TYPE "LBP_typeAxisX"
TITLE = Axis interface / Interface d'axe
// User data type for blocks LBP_Axis1 [DB31] .. LBP_Axis31 [DB61] / Type de données utilisateur pour les blocs LBP_Axis1 [DB31] .. LBP_Axis31 [DB61]
   STRUCT
      A_FD_OR : Byte;   // Feedrate override / Correction d'avance
      A_DriveEnable : Bool;   // Drive test movement enable / Débloquer le déplacement pour test d'entraînement
      A_AckFixedStop : Bool;   // Acknowledge fixed stop reached / Acquittement accostage de butée
      A_SensorFixedStop : Bool;   // Sensor fixed stop / Détecteur butée
      A_ASpDisable : Bool;   // Axis/spindle disable / Désactiver axe/broche
      A_Follow_upMode : Bool;   // Follow-up mode / Mode poursuite
      A_PosMeas1 : Bool;   // Position measuring system 1 / Système de mesure de position 1
      A_PosMeas2 : Bool;   // Position measuring system 2 / Système de mesure de position 2
      A_ORactive : Bool;   // Override active / Correction active
      A_SWCam : Bool;   // SW cam activation / Activation came logicielle
      A_ContrEnable : Bool;   // Controller enable / Activer la commande
      A_DelDTGSpReset : Bool;   // Delete distance to go/Spindle-Reset / Effacer la distance restante à parcourir / Reset broche
      A_Clamp : Bool;   // Clamping in progress / Serrage en cours
      A_RefVal1 : Bool;   // Reference point value 1 / Valeur de point de référence 1
      A_RefVal2 : Bool;   // Reference point value 2 / Valeur de point de référence 2
      A_RefVal3 : Bool;   // Reference point value 3 / Valeur de point de référence 3
      A_RefVal4 : Bool;   // Reference point value 4 / Valeur de point de référence 4
      A_ExtZO : Bool;   // Import external ZO / Importer ZO externes
      A_EnabTravFixedStop : Bool;   // Enable travel to fixed stop / Activer déplacement pour accostage de butée
      A_FixedFD1 : Bool;   // Activate fixed feedrate 1 / Activer l'avance fixe 1
      A_FixedFD2 : Bool;   // Activate fixed feedrate 2 / Activer l'avance fixe 2
      A_FixedFD3 : Bool;   // Activate fixed feedrate 3 / Activer l'avance fixe 3
      A_FixedFD4 : Bool;   // Activate fixed feedrate 4 / Activer l'avance fixe 4
      A_VelocSpeedLimit : Bool;   // Velocity/spindle speed limitation / Limitation vitesse / vitesse de broche
      A_PrgtestAxRel : Bool;   // Program test axis/spindle release / Débloquer test de programme axe/broche
      A_HW1 : Bool;   // Activate handwheel 1 / Activer manivelle 1
      A_HW2 : Bool;   // Activate handwheel 2 / Activer manivelle 2
      A_HW3 : Bool;   // Activate handwheel 3 / Activer manivelle 3
      A_FDSpStop : Bool;   // Feed stop/spindle stop / Arrêt avance / arrêt broche
      A_Disable : Bool;   // Traversing key disable / Désactiver la touche de déplacement
      A_RapidTrOR : Bool;   // Rapid traverse override / Correction marche rapide
      A_Minus : Bool;   // Traversing key minus / Touche de déplacement moins
      A_Plus : Bool;   // Traversing key plus / Touche de déplacement plus
      A_INC1 : Bool;   // INC1
      A_INC10 : Bool;   // INC10
      A_INC100 : Bool;   // INC100
      A_INC1000 : Bool;   // INC1000
      A_INC10000 : Bool;   // INC10000
      A_INCVar : Bool;   // INC variable / Variable INC
      A_ContManTravel : Bool;   // Continuous manual travel / Mode manuel continu
      f5_7 : Bool;
      A_OEMAxis : Byte;   // OEM axis signals / Signaux des axes OEM
      A_InvHWDirOfRot : Bool;   // Inverting handwheel direction of rotation / Inverser sens de rotation manivelle
      f7_1 : Bool;
      f7_2 : Bool;
      f7_3 : Bool;
      f7_4 : Bool;
      f7_5 : Bool;
      f7_6 : Bool;
      f7_7 : Bool;
      A_NCASpChanA : Bool;   // Assign NC axis/spindle channel A / Affecter axe/broche CN au canal A
      A_NCASpChanB : Bool;   // Assign NC axis/spindle channel B / Affecter axe/broche CN au canal B
      A_NCASpChanC : Bool;   // Assign NC axis/spindle channel C / Affecter axe/broche CN au canal C
      A_NCASpChanD : Bool;   // Assign NC axis/spindle channel D / Affecter axe/broche CN au canal D
      A_NCASpStrobe : Bool;   // Activation of assignment with pos. edge / Activation de l'affection sur font montant
      f8_5 : Bool;
      f8_6 : Bool;
      A_PLCASp : Bool;   // Request PLC axis/spindle / Demander axe/broche AP
      A_Para_A : Bool;   // Parameter block servo A / Bloc de paramètres servo A
      A_Para_B : Bool;   // Parameter block servo B / Bloc de paramètres servo B
      A_Para_C : Bool;   // Parameter block servo C / Bloc de paramètres servo C
      A_LockParSetDef : Bool;   // Lock parameter set definition from NC / Bloquer la définition de jeu de paramètre depuis CN
      f9_4 : Bool;
      f9_5 : Bool;
      f9_6 : Bool;
      f9_7 : Bool;
      A_REPOSDelay : Bool;   // REPOS DELAY
      f10_1 : Bool;
      f10_2 : Bool;
      f10_3 : Bool;
      f10_4 : Bool;
      f10_5 : Bool;
      f10_6 : Bool;
      f10_7 : Bool;
      A_StartBrakeTest : Bool;   // Start brake test / Démarrer test de frein
      f11_1 : Bool;
      f11_2 : Bool;
      f11_3 : Bool;
      f11_4 : Bool;
      f11_5 : Bool;
      f11_6 : Bool;
      f11_7 : Bool;
      A_HWLimitMinus : Bool;   // Hardware limit switch minus / Fin de course matériel moins
      A_HWLimitPlus : Bool;   // Hardware limit switch plus / Fin de course matériel plus
      A_SWLimit2Minus : Bool;   // 2nd software limit switch minus / 2e fin de course logiciel moins
      A_SWLimit2Plus : Bool;   // 2nd software limit switch plus / 2e fin de course logiciel plus
      A_ModuloLimitEn : Bool;   // Modulo limit enabled / Limite modulo activée
      f12_5 : Bool;
      f12_6 : Bool;
      A_DelayRef : Bool;   // Delay reference point approach / Retarder l'accostage de point de référence
      A_JogFixPPos0 : Bool;   // JogFixPointPos 0
      A_JogFixPPos1 : Bool;   // JogFixPointPos 1
      A_JogFixPPos2 : Bool;   // JogFixPointPos 2
      A_JogToPos : Bool;   // Jog to position / Mode JOG vers position
      f13_4 : Bool;
      f13_5 : Bool;
      f13_6 : Bool;
      f13_7 : Bool;
      A_ProgtestSuppress : Bool;   // Program test to suppress / Inhiber test de programme
      A_ProgtestActivate : Bool;   // Activate program test / Activer test de programme
      f14_2 : Bool;
      f14_3 : Bool;
      f14_4 : Bool;
      f14_5 : Bool;
      f14_6 : Bool;
      f14_7 : Bool;
      f15 : Byte;
      A_ActGearA : Bool;   // Current gear stage A / Rapport de transmission actuel A
      A_ActGearB : Bool;   // Current gear stage B / Rapport de transmission actuel B
      A_ActGearC : Bool;   // Current gear stage C / Rapport de transmission actuel C
      A_GearChangeOv : Bool;   // Gear has changed over / Réducteur a changé de rapport
      A_Sp1Syn : Bool;   // Re-synchronize spindle 1 / Resynchroniser broche 1
      A_Sp2Syn : Bool;   // Re-synchronize spindle 2 / Resynchroniser broche 2
      A_NoMonitorGear : Bool;   // No monitoring when changing gear / Aucune surveillance pendant le changement de rapport de réducteur
      A_DeleteS : Bool;   // Delete S value / Supprimer la valeur S
      A_FD_ORSp : Bool;   // Feedrate override for spindle valid / Correction d'avance pour broche valide
      f17_1 : Bool;
      f17_2 : Bool;
      f17_3 : Bool;
      A_Sp1SynP : Bool;   // Re-synchronize spindle 1 for positioning / Resynchroniser broche 1 pour positionnement
      A_Sp2SynP : Bool;   // Re-synchronize spindle 2 for positioning / Resynchroniser broche 2 pour positionnement
      A_M3M4Inv : Bool;   // Invert M3/M4 / Inverser M3/M4
      f17_7 : Bool;
      f18_0 : Bool;
      f18_1 : Bool;
      f18_2 : Bool;
      f18_3 : Bool;
      A_OscilPLC : Bool;   // Oscillation via PLC / Oscillation via AP
      A_OscilSpeed : Bool;   // Enable Oscillation / Activer oscillation
      A_SetRotDirectRight : Bool;   // Setpoint osci. direct. right / Consigne sens d'oscillation à droite
      A_SetRotDirectLeft : Bool;   // Setpoint osci. direct. left / Consigne sens d'oscillation à gauche
      A_SpOR : Byte;   // Spindle override / Correction broche
      f20_0 : Bool;
      A_RUEncQuStop : Bool;   // Run-up encoder quick stop / Générateur de rampe Arrêt rapide
      f20_2 : Bool;
      A_SpeedSetpSmooth : Bool;   // Speed setpoint smoothing / Lissage consigne de vitesse
      f20_4 : Bool;
      A_HoldBrakeToOpen : Bool;   // Holding brake open / Frein à l'arrêt desserré
      f20_6 : Bool;
      f20_7 : Bool;
      A_ParA : Bool;   // Parameter set selection A / Jeux de paramètres sélection A
      A_ParB : Bool;   // Parameter set selection B / Jeux de paramètres sélection B
      A_ParC : Bool;   // Parameter set selection C / Jeux de paramètres sélection C
      A_MotA : Bool;   // Motor selection A / Sélection moteur A
      A_MotB : Bool;   // Motor selection B / Sélection moteur B
      A_MotOK : Bool;   // Motor selected / Moteur sélectionné
      A_IntegratDisable : Bool;   // N controller integrator disable / Commande N Désactiver intégrateur
      A_PulseEnable : Bool;   // Pulse enable / Activer impulsions
      f22_0 : Bool;
      f22_1 : Bool;
      f22_2 : Bool;
      f22_3 : Bool;
      f22_4 : Bool;
      f22_5 : Bool;
      f22_6 : Bool;
      f22_7 : Bool;
      f23_0 : Bool;
      f23_1 : Bool;
      f23_2 : Bool;
      f23_3 : Bool;
      f23_4 : Bool;
      f23_5 : Bool;
      f23_6 : Bool;
      f23_7 : Bool;
      f24_0 : Bool;
      A_ControlAx : Bool;   // Control Axis / Axe pilote
      f24_2 : Bool;
      f24_3 : Bool;
      A_TorqComp : Bool;   // Torque compensation / Compensation de couple
      A_ChangSetpOutAss0 : Bool;   // Bit value for CTRLOUT_changed - Change setpoint output assignment / Valeur de bit pour CTRLOUT_changed - Modifier l'affectation de la sortie de consigne
      A_ChangSetpOutAss1 : Bool;   // Bit value for CTRLOUT_changed - Change setpoint output assignment / Valeur de bit pour CTRLOUT_changed - Modifier l'affectation de la sortie de consigne
      A_MS : Bool;   // Main/Sub: activate coupling / Maître/esclave : activer le couplage
      A_DynBComp : Bool;   // Dynamic backlash compensation activated / Compensation dynamique de jeu activée
      f25_1 : Bool;
      f25_2 : Bool;
      f25_3 : Bool;
      f25_4 : Bool;
      f25_5 : Bool;
      f25_6 : Bool;
      f25_7 : Bool;
      f26_0 : Bool;
      f26_1 : Bool;
      f26_2 : Bool;
      A_CompContr : Bool;   // Compensation controller On / Contrôleur de compensation MARCHE
      A_FollowAxOv : Bool;   // Enable following axis override / Activer la correction de l'axe asservi
      f26_5 : Bool;
      f26_6 : Bool;
      f26_7 : Bool;
      A_DEPMCS : Bool;   // Resume: DEPMCS / Continuer : DEPMCS
      A_DEPBCS : Bool;   // Resume: DEPBCS / Continuer : DEPBCS
      A_Corr : Bool;   // Resume: Corr / Continuer : corr
      A_HIAxMove : Bool;   // Resume: HIAxMove / Continuer : HIAxMove
      A_StopDEPMCS : Bool;   // Stop: DEPMCS / Arrêt : DEPMCS
      A_StopDEPBCS : Bool;   // Stop: DEPBCS / Arrêt : DEPBCS
      A_StopCorr : Bool;   // Stop: Corr / Arrêt : corr
      A_StopHIAxMove : Bool;   // Stop: HIAxMove / Arrêt : HIAxMove
      A_OscillAxExtRev : Bool;   // OscillAxExtReversal
      A_AxReset : Bool;   // AXRESET
      A_AxResume : Bool;   // AXRESUME
      A_SetRP : Bool;   // Set reversal point / Définir point d'inversion
      A_ChangeRP : Bool;   // Change reversal point / Modifier le point d'inversion
      A_StopRP : Bool;   // Stop at next reversal point / Arrêt sur point d'inversion suivant
      A_Stop : Bool;   // Stop / Arrêt
      A_PLCAxis : Bool;   // PLC checks axis / AP vérifie axe
      f29_0 : Bool;
      f29_1 : Bool;
      f29_2 : Bool;
      f29_3 : Bool;
      A_StartGantSynRun : Bool;   // Start gantry synchronization run / Démarrer l'opération de synchronisation Gantry
      A_NoAutoSync : Bool;   // No auto sync / Aucune sync auto
      f29_6 : Bool;
      f29_7 : Bool;
      A_StopSpindle : Bool;   // Stop spindle / Arrêt broche
      A_StartCW : Bool;   // Start spindle clockwise / Démarrer broche avec rotation horaire
      A_StartCCW : Bool;   // Start spindle counterclockwise / Démarrer broche avec rotation antihoraire
      A_AutoGearStep : Bool;   // Autom. gear step change / Chmnt. auto rapport transmission
      A_PosSpindle : Bool;   // Position spindle / Position de broche
      f30_5 : Bool;
      f30_6 : Bool;
      f30_7 : Bool;
      f31_0 : Bool;
      f31_1 : Bool;
      f31_2 : Bool;
      f31_3 : Bool;
      A_Resynchronize : Bool;   // Resynchronize / Resynchroniser
      A_DisSync : Bool;   // Disable synchronization / Désactiver la synchronisation
      A_Tracksync : Bool;   // Track synchronism / Tracer synchronisme
      A_DelSyncRunCorr : Bool;   // Deleting synchronous run correction / Suppression de la correction marche synchrone
      f32_0 : Bool;
      f32_1 : Bool;
      f32_2 : Bool;
      f32_3 : Bool;
      f32_4 : Bool;
      f32_5 : Bool;
      f32_6 : Bool;
      f32_7 : Bool;
      f33_0 : Bool;
      f33_1 : Bool;
      f33_2 : Bool;
      f33_3 : Bool;
      f33_4 : Bool;
      f33_5 : Bool;
      f33_6 : Bool;
      f33_7 : Bool;
      A_SI_SetpLimBit0 : Bool;   // Set point limitation Bit0 / Limitation de consigne Bit 0
      A_SI_SetpLimBit1 : Bool;   // Set point limitation Bit1 / Limitation de consigne Bit 1
      f34_2 : Bool;
      A_ActivateBrakeRampForSs2e : Bool;   // Brakes with NCK ramp on selection of SS2E (MD36959 MA_SAFE_BRAKE_RAMP_TIME) / Freinage avec rampe du NCK lors de la sélection de SS2E (MD36959 MA_SAFE_BRAKE_RAMP_TIME)
      f34_4 : Bool;
      f34_5 : Bool;
      f34_6 : Bool;
      f34_7 : Bool;
      f35 : Byte;
      f36 : Array[36..55] of Byte;
      A_FeedDriveCAxEng : Bool;   // Separate feed drive as C axis engaged / Entraînement d'avance séparé activé en tant qu'axe C
      A_SpSpeedDisp : Bool;   // Spindle speed display / Affichage vitesse de broche
      A_SpInsideClamp : Bool;   // Spindle inside clamping / Serrage interne broche
      f56_3 : Bool;
      f56_4 : Bool;
      f56_5 : Bool;
      f56_6 : Bool;
      f56_7 : Bool;
      f57 : Byte;
      f58 : Word;
      E_SpNA : Bool;   // Spindle/no axis / Broche / aucun axe
      E_NCU_Link : Bool;   // NCU_link active axis / NCU_link axe actif
      E_EncodFreq1 : Bool;   // Encoder limit frequency 1 exceeded / Fréquence limite capteur 1 dépassée
      E_EncodFreq2 : Bool;   // Encoder limit frequency 2 exceeded / Fréquence limite capteur 2 dépassée
      E_RefSyn1 : Bool;   // Referenced/synchronized 1 / Référencé/synchronisé 1
      E_RefSyn2 : Bool;   // Referenced/synchronized 2 / Référencé/synchronisé 2
      E_ExactCoarse : Bool;   // Position reached with exact stop coarse / Position atteinte avec arrêt précis approx.
      E_ExactFine : Bool;   // Position reached with exact stop fine / Position atteinte avec arrêt précis fin
      E_TravRequ : Bool;   // Travel request / Demande de déplacement
      E_AxialAlarm : Bool;   // Axial alarm / Alarme d'axe
      E_AxisReady : Bool;   // Axis ready / Axe prêt
      E_Follow_upMode : Bool;   // Follow-up mode active / Mode poursuite actif
      E_Stat : Bool;   // Axis/spindle stationary (n<nmin) / Axe/broche à l'arrêt (n<nmin)
      E_PositContr : Bool;   // Position controller active / Commande de positionnement active
      E_SpeedContr : Bool;   // Speed controller active / Régulateur de vitesse actif
      E_CurrentContr : Bool;   // Current controller active / Commande actuelle active
      E_SWCam : Bool;   // Software cams active / Came logicielle active
      E_HWOverlay : Bool;   // Handwheel overlay active / Superposition manivelle actif
      E_RevFD : Bool;   // Revolutional feedrate active / Avance par tour active
      E_MeasAct : Bool;   // Measuring active / Mesurage actif
      E_ActTravFStop : Bool;   // Activate travel to fixed stop / Activer déplacement pour accostage de butée
      E_FixedStop : Bool;   // Fixed stop reached / Butée atteinte
      E_ForceFixedStop : Bool;   // Force fixed stop limited / Force butée limitée
      E_AxContainerRot : Bool;   // Axis container rotation active / Conteneur d'axe Rotation activée
      E_AxReset : Bool;   // Axis reset done / Reset axe effectué
      E_PLCCtrlAx : Bool;   // PLC controlled axis / Axe commandé par AP
      E_AxStop : Bool;   // Axis stop active / Arrêt d'axe actif
      E_AxSpDisable : Bool;   // Axis/spindle disable active / Désactivation axe/broche active
      E_StopDEPMCS : Bool;   // Stop DEPMCS active / Arrêt DEPMCS actif
      E_StopDEPBCS : Bool;   // Stop DEPBCS active / Arrêt DEPBCS actif
      E_StopCorr : Bool;   // Stop Corr active / Arrêt corr actif
      E_StopHIAxMove : Bool;   // Stop HIAxMove active / Arrêt HIAxMove actif
      E_HW1 : Bool;   // Handwheel 1 active / Manivelle 1 active
      E_HW2 : Bool;   // Handwheel 2 active / Manivelle 2 active
      E_HW3 : Bool;   // Handwheel 3 active / Manivelle 3 active
      f64_3 : Bool;
      E_TReqMinus : Bool;   // Travel request minus / Demande de déplacement moins
      E_TReqPlus : Bool;   // Travel request plus / Demande de déplacement plus
      E_TCMinus : Bool;   // Traverse command minus / Instruction de déplacement moins
      E_TCPlus : Bool;   // Traverse command plus / Instruction de déplacement plus
      E_INC1 : Bool;   // INC1
      E_INC10 : Bool;   // INC10
      E_INC100 : Bool;   // INC100
      E_INC1000 : Bool;   // INC1000
      E_INC10000 : Bool;   // INC10000
      E_INCVar : Bool;   // INC variable / Variable INC
      E_ContManTravelAct : Bool;   // Continuous manual travel active / Mode manuel continu actif
      f65_7 : Bool;
      E_OEMAxis : Byte;   // OEM axis signals / Signaux des axes OEM
      E_InvHWDirOfRot : Bool;   // Handwheel direction of rotation invert actively / Inverser activement sens manivelle
      f67_1 : Bool;
      f67_2 : Bool;
      f67_3 : Bool;
      f67_4 : Bool;
      f67_5 : Bool;
      f67_6 : Bool;
      f67_7 : Bool;
      E_NCASpChanA : Bool;   // NC axis/spindle in channel A / Axe/broche CN dans canal A
      E_NCASpChanB : Bool;   // NC axis/spindle in channel B / Axe/broche CN dans canal B
      E_NCASpChanC : Bool;   // NC axis/spindle in channel C / Axe/broche CN dans canal C
      E_NCASpChanD : Bool;   // NC axis/spindle in channel D / Axe/broche CN dans canal D
      E_PLCType : Bool;   // New type requested by PLC / Nouveau type demandé de l'AP
      E_ChPoss : Bool;   // Change axis possible / Modification d'axe possible
      E_NeutrASp : Bool;   // Neutral axis/spindle / Axe/broche neutre
      E_PLCASp : Bool;   // PLC axis/spindle / Axe/broche AP
      E_ParS_A : Bool;   // Parameter block servo A / Bloc de paramètres servo A
      E_ParS_B : Bool;   // Parameter block servo B / Bloc de paramètres servo B
      E_ParS_C : Bool;   // Parameter block servo C / Bloc de paramètres servo C
      E_NCUNumLink_3 : Bool;
      E_NCUNumLink_4 : Bool;
      E_NCUNumLink_5 : Bool;
      E_NCUNumLink_6 : Bool;
      E_NCUNumLink_7 : Bool;
      E_ReposSh : Bool;   // REPOS shift / REPOS Décalage
      E_ReposShValid : Bool;   // REPOS shift valid / REPOS Décalage valide
      E_ReposDelayQuit : Bool;   // REPOS delay quit / REPOS Terminer temporisation
      f70_3 : Bool;
      f70_4 : Bool;
      E_SI_Drv_SICSCC : Bool;   // DRV-Safety Integrated with SIC/SCC active / DRV Safety Integrated avec SIC/SCC actif
      E_SI_Drv_Parameterized : Bool;   // Drive based Safety Intergated (SI) function enabled (at least one function in parameter "p9501" or "p9601" is parameterized) / Fonction Drive based Safety Integrated (SI) débloquée (au moins une fonction est paramétrée dans le paramètre "p9501" ou "p9601")
      f70_7 : Bool;
      E_BrakeTest : Bool;   // Brake test active / Test de frein actif
      f71_1 : Bool;
      f71_2 : Bool;
      f71_3 : Bool;
      E_POS_RESTORED1 : Bool;   // POS_RESTORED 1
      E_POS_RESTORED2 : Bool;   // POS_RESTORED 2
      f71_6 : Bool;
      E_PLCAxDedic : Bool;   // PLC axis dedicated / Axe AP dédié
      E_MMC_REPOSDelay : Bool;   // HMI REPOS DELAY
      f72_1 : Bool;
      f72_2 : Bool;
      f72_3 : Bool;
      f72_4 : Bool;
      f72_5 : Bool;
      f72_6 : Bool;
      f72_7 : Bool;
      f73 : Byte;
      f74_0 : Bool;
      f74_1 : Bool;
      f74_2 : Bool;
      f74_3 : Bool;
      E_ModLimEnAct : Bool;   // Modulo limit enabled active / Limite modulo activée actif
      f74_5 : Bool;
      f74_6 : Bool;
      f74_7 : Bool;
      E_JogFixPPos0Act : Bool;   // JogFixPointPos 0 active / JogFixPointPos 0 activé
      E_JogFixPPos1Act : Bool;   // JogFixPointPos 1 active / JogFixPointPos 1 activé
      E_JogFixPPos2Act : Bool;   // JogFixPointPos 2 active / JogFixPointPos 2 activé
      E_JogFixPPos0 : Bool;   // JogFixPointPos 0 reached / JogFixPointPos 0 atteint
      E_JogFixPPos1 : Bool;   // JogFixPointPos 1 reached / JogFixPointPos 1 atteint
      E_JogFixPPos2 : Bool;   // JogFixPointPos 2 reached / JogFixPointPos 2 atteint
      E_JogToPos : Bool;   // Jog to position active / Mode JOG vers position actif
      E_JogPos : Bool;   // Jog position reached / Position JOG atteinte
      E_ScratchPulse : Bool;   // Scratch pulse
      f76_1 : Bool;
      f76_2 : Bool;
      f76_3 : Bool;
      E_PathAxis : Bool;   // Path axis / Axe d'interpolation
      E_PosAxis : Bool;   // Positioning axis / Axe de positionnement
      E_IndexAxisPos : Bool;   // Indexing axis in position / Axe indexé en position
      E_CurvePos : Bool;   // Curve axis in position / Axe de contournage en position
      E_CollCheckRedSpeed : Bool;   // Reduced speed of Collisions Check / Vitesse réduite du contrôle de collision
      f77_1 : Bool;
      f77_2 : Bool;
      f77_3 : Bool;
      f77_4 : Bool;
      f77_5 : Bool;
      f77_6 : Bool;
      f77_7 : Bool;
      E_FPosAxis : Real;   // F function (REAL format) for positioning axes / Fonction F (format REAL) pour axes de positionnement
      E_SetpGearA : Bool;   // Setpoint gear stage A / Consigne de rapport de transmission A
      E_SetpGearB : Bool;   // Setpoint gear stage B / Consigne de rapport de transmission B
      E_SetpGearC : Bool;   // Setpoint gear stage C / Consigne de rapport de transmission C
      E_GearChange : Bool;   // Gear changeover / Changement de rapport réducteur
      f82_4 : Bool;
      f82_5 : Bool;
      f82_6 : Bool;
      f82_7 : Bool;
      E_SpeedLimit : Bool;   // Speed limit exceeded / Limite de vitesse dépassée
      E_SetSpeedLimit : Bool;   // Setpoint speed limited / Consigne de vitesse limitée
      E_SetSpeedIncreased : Bool;   // Setpoint speed increased / Consigne de vitesse augmentée
      E_GeoMonit : Bool;   // Geometry monitoring / Surveillance de géométrie
      E_SupportAreaViol : Bool;   // Support area limits violated / Limites de la zone de support dépassées
      E_SetRange : Bool;   // Spindle in setpoint range / Broche dans la plage consigne
      E_SpeedMonit : Bool;   // Speed monitoring / Surveillance de vitesse
      E_ActRotRight : Bool;   // Actual rotation direction right / Sens de rotation actuel horaire
      E_ConstCuttSpeed : Bool;   // Const. cutting speed active / Vitesse de coupe constante active
      E_SUG : Bool;   // SUG active (grinding wheel surface speed) / VPM active (vitesse périphérique de meule)
      E_CLG : Bool;   // CLG active / CLG actif
      E_Tapping : Bool;   // Tapping without compensating chuck / Taraudage sans porte-taraud compensateur
      E_SyncMode : Bool;   // Synchronous mode spindle active / Mode broche synchrone actif
      E_PosMode : Bool;   // Positioning mode spindle active / Mode positionnement broche actif
      E_OscillMode : Bool;   // Oscillation mode spindle active / Mode oscillation broche actif
      E_ContrMode : Bool;   // Control mode spindle active / Mode de commande broche actif
      E_ToolDynLimit : Bool;   // Tool with dynamics limit / Outil avec limite dynamique
      f85_1 : Bool;
      f85_2 : Bool;
      f85_3 : Bool;
      f85_4 : Bool;
      E_SpInPosition : Bool;   // Spindle in position / Broche en position
      f85_6 : Bool;
      f85_7 : Bool;
      E_MFunct : Int;   // M function (INT) for spindle / Fonction M (INT) pour broche
      E_SFunct : Real;   // S function (REAL) for spindle / Fonction S (REAL) pour broche
      f92_0 : Bool;
      E_RUEncDisabl : Bool;   // Run-up encoder disable active / Blocage codeur de démarrage actif
      f92_2 : Bool;
      E_SpeedSetpSmooth : Bool;   // Speed setpoint smoothing active / Lissage consigne de vitesse actif
      E_RLIact : Bool;   // RLI active / RLI actif
      E_HoldBrakeOpened : Bool;   // Holding brake opened / Frein à l'arrêt desserré
      f92_6 : Bool;
      E_DriveRunEn : Bool;   // Drive run enabled / Déplacement entraînement activé
      E_ParA : Bool;   // Active parameter set A / Jeux de paramètres actif A
      E_ParB : Bool;   // Active parameter set B / Jeux de paramètres actif B
      E_ParC : Bool;   // Active parameter set C / Jeux de paramètres actif C
      E_MotA : Bool;   // Active motor A / Moteur actif A
      E_MotB : Bool;   // Active motor B / Moteur actif B
      E_MotOK : Bool;   // Drive ready / Entraînement prêt
      E_IntegratDisable : Bool;   // N controller integrator disabled / Commande N Intégrateur désactivé
      E_PulseEnable : Bool;   // Pulses enabled / Impulsions débloquées
      E_MTempWarn : Bool;   // Prewarning motor temperature / Avertissement température moteur
      E_HTempWarn : Bool;   // Prewarning heat sink temperature / Avertissement température radiateur
      E_RUComplete : Bool;   // Ramp-up complete / Démarrage terminé
      E_MdMdx : Bool;   // Md<Mdx
      E_NactNmin : Bool;   // nact<nmin
      E_NactNx : Bool;   // nact<nx
      E_NactNset : Bool;   // nact=nset
      E_Message : Bool;   // Variable message function 1 / Fonction de signalisation variable 1
      E_UDClessAlThreshold : Bool;   // UDC-link < alarm threshold / Lien UDC < seuil d'alarme
      E_DcVoltageAlarmAct : Bool;   // ESR: DC link voltage is below the specified minimum / AER : la tension du circuit intermédiaire est inférieure au minimum spécifié
      E_GeneratorOperationAct : Bool;   // ESR: generator operation is active / AER : le fonctionnement du générateur est actif
      E_SpeedBelowMin : Bool;   // ESR: actual speed is below specified minimum speed - axis is a generator axis / AER : la vitesse réelle est inférieure à la vitesse minimale spécifiée – l'axe est un axe de générateur
      E_Message2 : Bool;   // Variable message function 2 / Fonction de signalisation variable 2
      E_Message3 : Bool;   // Variable message function 3 / Fonction de signalisation variable 3
      f95_6 : Bool;
      E_I2TLimit : Bool;   // Power Section I2T limit / Partie puissance limite I2T
      f96_0 : Bool;
      E_AxisCtrl : Bool;   // Axis control active / Commande d'axe active
      E_MSFine : Bool;   // Main/Sub: speed difference is within the fine tolerance range / Maître/esclave : la différence de vitesse se situe dans la plage de tolérance fine
      E_MSCoarse : Bool;   // Main/Sub: speed difference is within the coarse tolerance range / Maître/esclave : la différence de vitesse se situe dans la plage de tolérance grossière
      E_MSCompContr : Bool;   // Main/Sub: torque compensatory controller is active / Maître/esclave : le régulateur de compensation de couple est actif
      E_BitValCtrlOutChang0 : Bool;   // Bit value for CTRLOUT_changed 0: Change setpoint output assignment / Valeur de CTRLOUT_changed 0 : modifier l'affectation de sortie de consigne
      E_BitValCtrlOutChang1 : Bool;   // Bit value for CTRLOUT_changed 1: Change setpoint output assignment / Valeur de CTRLOUT_changed 1 : modifier l'affectation de sortie de consigne
      E_MS : Bool;   // Main/Sub: coupling is active / Maître/esclave : le couplage est actif
      f97 : Byte;
      E_SyncronFine : Bool;   // Synchronism fine / Synchronisme fin
      E_SyncronCoarse : Bool;   // Synchronism coarse / Synchronisme approx
      E_ActValCoupling : Bool;   // Actual value coupling / Valeur réelle couplage
      f98_3 : Bool;
      E_OverlayMotion : Bool;   // Overlaid motion / Mouvement superposé
      E_SWL : Bool;   // Speed warning limit reached / Valeur limite d'alarme pour vitesse atteinte
      E_AWL : Bool;   // Acceleration warning limit reached / Valeur limite d'alarme pour accélération atteinte
      E_EmRetr : Bool;   // Emergency retraction active / Retrait d'urgence actif
      E_MasterSp : Bool;   // Generic coupling: spindle is leading spindle / Couplage générique : la broche est une broche pilote
      E_SlaveSp : Bool;   // Generic coupling: spindle is following spindle / Couplage générique : la broche est une broche asservie
      E_SyncRunCorrDOut : Bool;   // Synchronous run correction driven out / Correction synchronisme dépassée
      E_AxisAccel : Bool;   // Axis accelerated / Axe accéléré
      E_Sync : Bool;   // Synchronization active / Synchronisation active
      E_MSR : Bool;   // Max. speed reached / Vitesse max. atteinte
      E_MAR : Bool;   // Max. acceleration reached / Accélération max. atteinte
      f99_7 : Bool;
      f100_0 : Bool;
      f100_1 : Bool;
      E_OscillAxExtRev : Bool;   // OscillAxExt Reversal active / OscillAxExt Inversion active
      E_StopOscill : Bool;   // Oscillation cannot start / Impossible de démarrer oscillation
      E_ErrorOscill : Bool;   // Error during oscillation / Erreur lors de l'oscillation
      E_SparkOut : Bool;   // Spark-out active / Passes à lécher actives
      E_OscillMotion : Bool;   // Oscillation motion active / Mouvement d'oscillation actif
      E_Oscill : Bool;   // Oscillation active
      f101_0 : Bool;
      f101_1 : Bool;
      E_GantCOLimit : Bool;   // Gantry cut-off limit exceeded / Limite coupure axe Gantry atteinte
      E_GantWarn : Bool;   // Gantry warning limit exceeded / Gantry Limite d'alarme dépassée
      E_SynRunStart : Bool;   // Synchronization run ready to start / Synchronisme prêt à démarrer
      E_GantGroupSyn : Bool;   // Gantry grouping is synchronous / Groupage Gantry synchronisé
      E_GantLeadAxis : Bool;   // Gantry leading axis / Axe pilote Gantry
      E_GantAxis : Bool;   // Gantry axis / Axe Gantry
      E_DynBComp : Bool;   // Dynamic backlash compensation activated / Compensation dynamique de jeu activée
      f102_1 : Bool;
      f102_2 : Bool;
      E_ClampTolerance : Bool;   // Clamp tolerance exceeded / Tolérance de serrage d'axe dépassée
      f102_4 : Bool;
      E_PosMeas1 : Bool;   // Position measuring system 1 active / Système de mesure de position 1 actif
      E_PosMeas2 : Bool;   // Position measuring system 2 active / Système de mesure de position 2 actif
      f102_7 : Bool;
      E_SyncRunCorrIncl : Bool;   // Synchronous run correction is included / Correction synchronisme incluse
      f103_1 : Bool;
      f103_2 : Bool;
      f103_3 : Bool;
      E_Syncron2Fine : Bool;   // Synchronism fine / Synchronisme fin
      E_Syncron2Coarse : Bool;   // Synchronism coarse / Synchronisme approx
      f103_6 : Bool;
      f103_7 : Bool;
      E_AIAxis : Array[1..31] of Bool;   // Active infeed axis[1..31] / Axe de pénétration active [1..31]
      f108_0 : Bool;
      f108_1 : Bool;
      f108_2 : Bool;
      f108_3 : Bool;
      f108_4 : Bool;
      f108_5 : Bool;
      f108_6 : Bool;
      f108_7 : Bool;
      f109_0 : Bool;
      f109_1 : Bool;
      f109_2 : Bool;
      f109_3 : Bool;
      f109_4 : Bool;
      f109_5 : Bool;
      f109_6 : Bool;
      f109_7 : Bool;
      f110_0 : Bool;
      f110_1 : Bool;
      f110_2 : Bool;
      f110_3 : Bool;
      f110_4 : Bool;
      f110_5 : Bool;
      f110_6 : Bool;
      f110_7 : Bool;
      f111_0 : Bool;
      f111_1 : Bool;
      f111_2 : Bool;
      f111_3 : Bool;
      f111_4 : Bool;
      f111_5 : Bool;
      f111_6 : Bool;
      f111_7 : Bool;
      f112 : Byte;
      f113 : Byte;
      f114 : Byte;
      f115 : Byte;
      f116 : Byte;
      f117_0 : Bool;
      f117_1 : Bool;
      f117_2 : Bool;
      f117_3 : Bool;
      f117_4 : Bool;
      f117_5 : Bool;
      f117_6 : Bool;
      f117_7 : Bool;
      f118 : DWord;
      f122 : DWord;
      f126 : Word;   // Internal / Interne
      E_MMC_ProgtestSuppress : Bool;   // HMI->PLC: Suppress program test / HMI ->AP : inhiber test de programme
      E_MMC_ProgtestActivate : Bool;   // HMI->PLC: Activate program test / HMI ->AP : activer test de programme
      f128_2 : Bool;
      f128_3 : Bool;
      f128_4 : Bool;
      f128_5 : Bool;
      f128_6 : Bool;
      f128_7 : Bool;
      f129 : Byte;
      E_FormatBit0DDS : Bool;   // Bit 0 for drive data set switchover (DDS) / Bit 0 pour la commutation du jeu de paramètres d'entraînement (DDS)
      E_FormatBit1DDS : Bool;   // Bit 1 for drive data set switchover (DDS) / Bit 1 pour la commutation du jeu de paramètres d'entraînement (DDS)
      E_FormatBit2DDS : Bool;   // Bit 2 for drive data set switchover (DDS) / Bit 2 pour la commutation du jeu de paramètres d'entraînement (DDS)
      E_FormatBit3DDS : Bool;   // Bit 3 for drive data set switchover (DDS) / Bit 3 pour la commutation du jeu de paramètres d'entraînement (DDS)
      E_FormatBit4DDS : Bool;   // Bit 4 for drive data set switchover (DDS) / Bit 4 pour la commutation du jeu de paramètres d'entraînement (DDS)
      f130_5 : Bool;
      f130_6 : Bool;
      E_MDS_DDS_InterfacesValid : Bool;   // Motor and drive data set interfaces invalid / Jeux de paramètres moteur et d'entraînement Interfaces valides
      f131 : Byte;
      E_SensorAv : Bool;   // Sensors available / Capteurs disponibles
      E_S1aMeasARod : Bool;   // Sensor S1: analogous measurement position of actuating rod / Capteur S1 : position de mesure analogique de la tige d'actionnement
      f132_2 : Bool;
      f132_3 : Bool;
      E_S4dPistonStopP : Bool;   // Sensor S4: digital value piston stop position / Capteur S4 : valeur numérique position d'arrêt piston
      E_S5dAngleShaft : Bool;   // Sensor S5: digital value angle situation shaft / Capteur S5 : valeur numérique position angulaire arbre
      E_S6Temp : Bool;   // Sensor S6: temperature / Capteur S6 : température
      f132_7 : Bool;
      f133 : Byte;
      E_ClampingState : Int;   // State of the clamping system / État du système de serrage
      E_AnalogSensor : Int;   // Analog sensor on the motor / Capteur analogique sur moteur
      f138_0 : Bool;
      f138_1 : Bool;
      f138_2 : Bool;
      f138_3 : Bool;
      E_S4PistonStopP : Bool;   // Sensor S4: piston stop position / Capteur S4 : position d'arrêt piston
      E_S5AngleShaft : Bool;   // Sensor S5: angle situation shaft / Capteur S5 : position angulaire arbre
      f138_6 : Bool;
      f138_7 : Bool;
      f139 : Byte;
      SCC : Struct   // PLC to Drive (SCC) / AP vers entraînement (SCC)
         CW1 : Struct
            TeststopStart : Bool;   // Test stops for extended functions / Stops pour test pour fonctions étendues
            res140_1 : Bool;
            res140_2 : Bool;
            res140_3 : Bool;
            res140_4 : Bool;
            CloseBrake : Bool;   // Close internal Brake / Serrer le frein interne
            res140_6 : Bool;
            res140_7 : Bool;
            res141 : Byte;
         END_STRUCT;
         CW3 : Struct
            res142 : Byte;
            SelectionSBT : Bool;   // Selection: safe brake test / Sélection : test de frein sûr
            BT_Start : Bool;   // Start: brake test / Démarrage : test de frein
            Brake_1_2 : Bool;   // Brake test with brake 1 or 2 / Test de frein avec frein 1 ou 2
            DirOfROT : Bool;   // Direction of rotation / Sens de rotation
            Testseq_1_2 : Bool;   // Test sequence 1 or 2 / Séquence de test 1 ou 2
            BrakeClosed : Bool;   // Feedback external brake / Signalisation en retour frein externe
            res143_6 : Bool;
            res143_7 : Bool;
         END_STRUCT;
      END_STRUCT;
      res144_163 : Array[144..163] of Byte;
      SIC : Struct   // Drive to PLC (SIC) / Entraînement vers AP (SIC)
         SW1 : Struct
            SLA_Sel : Bool;   // Safely Limited Acceleration selected / Accélération limitée sûre sélectionnée
            SLS_LimBit0_Sel : Bool;   // Safely-Limited Speed: limit Bit0 selected / Vitesse limitée sûre : limite bit0 sélectionnée
            SLS_LimBit1_Sel : Bool;   // Safely-Limited Speed: limit Bit1 selected / Vitesse limitée sûre : limite bit1 sélectionnée
            res164_3 : Bool;
            res164_4 : Bool;
            res164_5 : Bool;
            ESR_Req : Bool;   // Extended Stop and Retract requested / Arrêt étendu et retrait demandé
            SF_Message_Act : Bool;   // Safety error active / Erreur de sécurité active
            STO_Act : Bool;   // Safe torque off: active / Suppression sûre du couple : active
            SS1_Act : Bool;   // Safe Stop1: active / Stop sûr 1 : actif
            SS2_Act : Bool;   // Safe Stop2: active / Stop sûr 2 : actif
            SOS_Act : Bool;   // Safe Operating Stop: active / Arrêt de fonctionnement sûr : actif
            SLS_Act : Bool;   // Safely-Limited Speed: active / Vitesse limitée sûre : active
            SOS_Sel : Bool;   // Safe Operating Stop: selected / Arrêt de fonctionnement sûr : sélectionné
            SLS_Sel : Bool;   // Safely-Limited Speed: selected / Vitesse limitée sûre : sélectionnée
            InternalEvent : Bool;   // Safety error with Stop A active / Erreur de sécurité avec butée A active
         END_STRUCT;
         SW2 : Struct
            SDI_P_Sel : Bool;   // Safe direction positive: selected / Direction sûre positive : sélectionnée
            SDI_N_Sel : Bool;   // Safe direction negative: selected / Direction sûre négative : sélectionnée
            res166_2 : Bool;
            res166_3 : Bool;
            TestStopAct : Bool;   // Test stop active / Stop pour test actif
            TestStopReq : Bool;   // Test stop requested / Stop pour test demandé
            res166_6 : Bool;
            res166_7 : Bool;
            res167_0 : Bool;
            res167_1 : Bool;
            res167_2 : Bool;
            res167_3 : Bool;
            SLP_LimBit0_Sel : Bool;   // Safely-Limited Position: limit Bit0 selected / Position limitée sûre : limite bit0 sélectionnée
            res167_5 : Bool;
            res167_6 : Bool;
            SLP_Sel : Bool;   // Safely-Limited Position: selected / Position limitée sûre : sélectionnée
         END_STRUCT;
         V_Limit_B : DInt;   // Setpoint speed limit effective / Limite de consigne de vitesse active
         SW3 : Struct
            res172_0 : Bool;
            res172_1 : Bool;
            res172_2 : Bool;
            SS2E_ACTIVE : Bool;   // SS2E active / SS2E actif
            SS2ESR : Bool;   // SS2ESR active / SS2ESR actif
            res172_5 : Bool;
            AcceptSLPAct : Bool;   // Acceptance test Safely-Limited Position active / Essai de réception position limitée sûre : actif
            AcceptTestSel : Bool;   // Acceptance test selected / Essai de réception sélectionné
            SBT_Sel : Bool;   // Safety break test: selected / Test de frein de sécurité : sélectionné
            SetpSettingDrive : Bool;   // Setpoint input is in the drive during the SBT / L'entrée de consigne est dans l'entraînement pendant le SBT
            Brake_1_2 : Bool;   // Test with brake 1 or 2 / Test avec frein 1 ou 2
            BT_Act : Bool;   // Brake test: active / Test de frein : actif
            BT_OK : Bool;   // Brake test: OK / Test de frein : OK
            BT_Finished : Bool;   // Brake test: finished / Test de frein : terminé
            BrakeReq : Bool;   // External brake close requested / Serrage de frein externe demandé
            SignLoadTorque : Bool;   // Sign of load torque is negative / Signe couple de charge négatif
         END_STRUCT;
      END_STRUCT;
      res174_187 : Array[174..187] of Byte;
      CW7 : Struct
         ReservedBit08 : Bool;
         ReservedBit09 : Bool;
         ReservedBit10 : Bool;
         ReservedBit11 : Bool;
         ReservedBit12 : Bool;
         ReservedBit13 : Bool;
         ReservedBit14 : Bool;
         ReservedBit15 : Bool;
         A_DisablePowerReduction : Bool;   // DYNEGMA: disable power reduction / DYNEGMA : désactiver la réduction de puissance
         A_DisableCurrReduction : Bool;   // Motor overtemperature: disable current reduction / Surchauffe du moteur : désactiver la réduction de puissance
         ReservedBit02 : Bool;
         ReservedBit03 : Bool;
         ReservedBit04 : Bool;
         ReservedBit05 : Bool;
         ReservedBit06 : Bool;
         ReservedBit07 : Bool;
      END_STRUCT;
      SW7 : Struct
         E_EncMaintenanceRequired : Bool;   // Encoder maintenance required / Maintenance du codeur requise
         ReservedBit09 : Bool;
         ReservedBit10 : Bool;
         ReservedBit11 : Bool;
         ReservedBit12 : Bool;
         ReservedBit13 : Bool;
         ReservedBit14 : Bool;
         ReservedBit15 : Bool;
         E_TorqueLimited : Bool;   // DYNEGMA: torque limited / DYNEGMA : couple limité
         E_CurrReductionActive : Bool;   // Motor overtemperature: current reduction active / Surchauffe du moteur : réduction de puissance active
         E_MotorTempModelAlarm : Bool;   // Motor overtemperature: motor temperature model alarm active / Surchauffe du moteur : alarme de modèle thermique du moteur active
         E_PolePosIdentPassed : Bool;   // Pole position identification with encoder successfully carried out / Identification de la position des pôles avec codeur effectuée avec succès
         ReservedBit04 : Bool;
         ReservedBit05 : Bool;
         E_AndConditionFulfilled : Bool;   // AND logic operation: condition fulfilled / Opération logique ET : condition remplie
         E_OrConditionFulfilled : Bool;   // OR logic operation: condition fulfilled / Opération logique OU : condition remplie
      END_STRUCT;
   END_STRUCT;
END_TYPE

TYPE "LBP_typeChanX"
TITLE = Channel interface / Interface de canal
// User data type for blocks LBP_Chan1 [DB21] .. LBP_Chan10 [DB30] / Type de données utilisateur pour les blocs LBP_Chan1 [DB21] .. LBP_Chan10 [DB30]
   STRUCT
      f0_0 : Bool;
      f0_1 : Bool;
      f0_2 : Bool;
      A_DRF : Bool;   // Activate DRF / Activer DRF
      A_SBL : Bool;   // Activate single block / Activer bloc par bloc
      A_M01 : Bool;   // Activate M01 / Activer M01
      A_DRY : Bool;   // Activate dry run feedrate / Activer avance marche d'essai
      f0_7 : Bool;
      A_Ref : Bool;   // Activate referencing / Activer référencement
      A_ProtZone : Bool;   // Enable protection zones / Activer zones de protection
      A_SynOff : Bool;   // Synchronous action off / Action synchrone désactivée
      A_TM_TimOut : Bool;   // Activate time-out (TM) / Activer timeout (TM)
      A_CLC_Stop : Bool;   // CLC stop / Stop CLC
      A_CLC_OR : Bool;   // CLC override / Correction CLC
      A_PLC_ActCompl : Bool;   // PLC action completed / Action AP terminée
      A_ProgTest : Bool;   // Activate program test / Activer test de programme
      A_SKP0 : Bool;   // Activate skip block \0 / Activer ignorer bloc \0
      A_SKP1 : Bool;   // Activate skip block \1 / Activer ignorer bloc \1
      A_SKP2 : Bool;   // Activate skip block \2 / Activer ignorer bloc \2
      A_SKP3 : Bool;   // Activate skip block \3 / Activer ignorer bloc \3
      A_SKP4 : Bool;   // Activate skip block \4 / Activer ignorer bloc \4
      A_SKP5 : Bool;   // Activate skip block \5 / Activer ignorer bloc \5
      A_SKP6 : Bool;   // Activate skip block \6 / Activer ignorer bloc \6
      A_SKP7 : Bool;   // Activate skip block \7 / Activer ignorer bloc \7
      A_StrokEnab : Bool;   // Stroke enable / Activer course
      A_ManStrokEnab : Bool;   // Manual stroke enable / Activation manuelle de la course
      A_StrokSup : Bool;   // Stroke suppression / Inhibition de course
      A_StrokDelayed : Bool;   // Stroke delayed / Course retardée
      A_StrokStop : Bool;   // Stroke not operating / Course inopérante
      A_ManRelStroke2 : Bool;   // Manual release of stroke 2 / Déblocage manuel de la course 2
      A3_6 : Bool;
      A3_7 : Bool;
      A_FD_OR : Byte;   // Feedrate override / Correction d'avance
      A_RT_OR : Byte;   // Rapid traverse override / Correction marche rapide
      A_FDdisable : Bool;   // Feed disable / Désactiver avance
      A_RIdisable : Bool;   // Read-in disable / Désactiver importation
      A_DeleteDTG : Bool;   // Delete distance to go / Effacer la distance restante à parcourir
      A_SP_Clear : Bool;   // Delete UP number of passes / Supprimer nombre UP de passes
      A_ProgAbort : Bool;   // Program level abort / Abandon niveau de programme
      A_F_Limit : Bool;   // Tool path feedrate limitation / Trajectoire d'outil limitation d'avance
      A_RT_ORA : Bool;   // Rapid traverse override active / Correction marche rapide active
      A_FD_ORA : Bool;   // Feedrate override active / Correction d'avance active
      A_NCStartDisabl : Bool;   // NC start disable / Désactiver Départ CN
      A_NCStart : Bool;   // NC start / Départ CN
      A_NCStopBlock : Bool;   // NC stop at block limit / Arrêt CN à la limite de bloc
      A_NCStop : Bool;   // NC stop / Arrêt CN
      A_NCStopASp : Bool;   // NC stop axes plus spindle / Arrêt CN axes et broche
      A_SuppStartLock : Bool;   // Suppress Start Lock / Inhiber blocage de démarrage
      A_CfgStopFunc : Bool;   // Activate configured stop function / Activer la fonction d'arrêt configuré
      A_Reset : Bool;   // Reset
      A_MRP : Array[1..10] of Bool;   // Activate machine-related protection zone [1..10] / Activer zone de protection référencée dans le SCM [1..10]
      A_CSP : Array[1..10] of Bool;   // Activate channel-specific protection zone [1..10] / Activer zone de protection spécifique au canal [1..10]
      A_Geo : Array[1..3] of Struct   // Control signals for geometry axis [1..3] / Signaux de commande pour axe géométrique [1..3]
         HW1 : Bool;   // Activate handwheel 1 / Activer manivelle 1
         HW2 : Bool;   // Activate handwheel 2 / Activer manivelle 2
         HW3 : Bool;   // Activate handwheel 3 / Activer manivelle 3
         FDStop : Bool;   // Feedrate stop / Arrêt avance
         Disabl : Bool;   // Traversing key disable / Désactiver la touche de déplacement
         RapidTrOR : Bool;   // Rapid traverse override / Correction marche rapide
         Minus : Bool;   // Traversing key minus / Touche de déplacement moins
         Plus : Bool;   // Traversing key plus / Touche de déplacement plus
         INC1 : Bool;   // INC 1
         INC10 : Bool;   // INC 10
         INC100 : Bool;   // INC 100
         INC1000 : Bool;   // INC 1000
         INC10000 : Bool;   // INC 10000
         INCVar : Bool;   // INC variable / Variable INC
         ContManTravel : Bool;   // Continuous manual travel / Mode manuel continu
         f1_7 : Bool;
         OEM : Byte;   // OEM signals / Signaux OEM
         InvHWDirOfRot : Bool;   // Invert handwheel direction of rotation / Inverser sens de rotation manivelle
         f3_1 : Bool;
         f3_2 : Bool;
         f3_3 : Bool;
         f3_4 : Bool;
         f3_5 : Bool;
         f3_6 : Bool;
         f3_7 : Bool;
      END_STRUCT;
      f24_0 : Bool;
      E_MMC_CfgStopFunc : Bool;   // HMI: configured stop function (CST) is selected / IHM : La fonction d'arrêt configuré (CST) est sélectionnée
      E_MMC_AtStopSetOvrZero : Bool;   // HMI: Set to 0% for stop override / IHM : à l'arrêt, régler la correction sur 0 %
      E_MMC_DRF : Bool;   // HMI DRF selected / HMI DRF sélectionné
      E_MMC_M01AssocNC : Bool;   // Select M01 associated with NC / Sélectionner M01 associé à CN
      E_MMC_M01 : Bool;   // HMI M01 selected / HMI M01 sélectionné
      E_MMC_DRY : Bool;   // HMI Dry-run feedrate selected / HMI Marche d'essai avance sélectionnée
      f24_7 : Bool;
      E_MMC_REPOSPM_0 : Bool;   // HMI REPOSPATHMODE 0
      E_MMC_REPOSPM_1 : Bool;   // HMI REPOSPATHMODE 1
      E_MMC_REPOSPM_2 : Bool;   // HMI REPOSPATHMODE 2
      E_MMC_FD_OR4RT_OR : Bool;   // HMI Feedrate override for rapid traverse selected / HMI Correction d'avance marche rapide sélectionnée
      E_MMC_REPOSMode : Bool;   // HMI REPOS MODE EDGE
      f25_5 : Bool;
      f25_6 : Bool;
      E_MMC_ProgTest : Bool;   // Program test selected / Test de programme sélectionné
      E_MMC_SKP0 : Bool;   // HMI skip block selected \0 / HMI Ignorer bloc sélectionné \0
      E_MMC_SKP1 : Bool;   // HMI skip block selected \1 / HMI Ignorer bloc sélectionné \1
      E_MMC_SKP2 : Bool;   // HMI skip block selected \2 / HMI Ignorer bloc sélectionné \2
      E_MMC_SKP3 : Bool;   // HMI skip block selected \3 / HMI Ignorer bloc sélectionné \3
      E_MMC_SKP4 : Bool;   // HMI skip block selected \4 / HMI Ignorer bloc sélectionné \4
      E_MMC_SKP5 : Bool;   // HMI skip block selected \5 / HMI Ignorer bloc sélectionné \5
      E_MMC_SKP6 : Bool;   // HMI skip block selected \6 / HMI Ignorer bloc sélectionné \6
      E_MMC_SKP7 : Bool;   // HMI skip block selected \7 / HMI Ignorer bloc sélectionné \7
      E_MMC_SKP8 : Bool;   // HMI skip block selected \8 / HMI Ignorer bloc sélectionné \8
      E_MMC_SKP9 : Bool;   // HMI skip block selected \9 / HMI Ignorer bloc sélectionné \9
      f27_2 : Bool;
      f27_3 : Bool;
      f27_4 : Bool;
      f27_5 : Bool;
      f27_6 : Bool;
      f27_7 : Bool;
      A_OEM : Byte;
      A_FixedFD1 : Bool;   // Activate fixed feedrate 1 / Activer l'avance fixe 1
      A_FixedFD2 : Bool;   // Activate fixed feedrate 2 / Activer l'avance fixe 2
      A_FixedFD3 : Bool;   // Activate fixed feedrate 3 / Activer l'avance fixe 3
      A_FixedFD4 : Bool;   // Activate fixed feedrate 4 / Activer l'avance fixe 4
      A_PTP_Travel : Bool;   // Activate PTP traversal / Activer déplacement PTP
      A_DisablWP_Counter : Bool;   // Deactivate workpiece counter / Désactiver compteur de pièces
      A_DisablWearMon : Bool;   // Deactivate wear monitoring / Désactiver surveillance d'usure
      A_DontDisablTool : Bool;   // Do not disable tool / Ne pas désactiver outil
      A_ContHW1 : Bool;   // Activate contour handwheel 1 / Activer manivelle de contour 1
      A_ContHW2 : Bool;   // Activate contour handwheel 2 / Activer manivelle de contour 2
      A_ContHW3 : Bool;   // Activate contour handwheel 3 / Activer manivelle de contour 3
      A_ContHWsim : Bool;   // Simulated contour handwheel on / Manivelle de contour simulée Marche
      A_ContHWneg : Bool;   // Contour handwheel neg. route / Manivelle de contour dépl. nég.
      A_NCKrelatedM01 : Bool;   // Activate NCK-related M01 / Activer M01 relatif à la NCK
      A_JOG_Circles : Bool;   // JOG in circles / JOG en cercles
      A_NoToolChangeCmd : Bool;   // No tool change commands / Aucun ordre de changement d'outil
      A_REPOSPM_0 : Bool;   // REPOSPATHMODE 0
      A_REPOSPM_1 : Bool;   // REPOSPATHMODE 1
      A_REPOSPM_2 : Bool;   // REPOSPATHMODE 2
      f31_3 : Bool;
      A_REPOSMode : Bool;   // REPOS MODE EDGE
      A_InvCHWDirOfRot : Bool;   // Inverting contour handwheel direction of rotation / Inversion du sens de rotation de la manivelle
      A_SKP8 : Bool;   // Activate skip block \8 / Activer ignorer bloc \8
      A_SKP9 : Bool;   // Activate skip block \9 / Activer ignorer bloc \9
      E_ExecExtern : Bool;   // Execution from external source active / Exécution à partir de source externe active
      f32_1 : Bool;
      f32_2 : Bool;
      E_ActBlock : Bool;   // Action block active / Bloc d'action actif
      E_BegBlock : Bool;   // Approach block active / Bloc d'accostage actif
      E_M01 : Bool;   // M0/M1 active / M0/M1 actif
      E_LastActBlock : Bool;   // Last action block active / Dernier bloc d'action actif
      f32_7 : Bool;
      E_Ref : Bool;   // Referencing active / Référencement actif
      E_OrieToolholder : Bool;   // Orientable toolholder active / Porte-outil orientable actif
      E_RevFD : Bool;   // Revolutional feedrate active / Avance par tour active
      E_HWOverlay : Bool;   // Handwheel override active / Correction manivelle active
      E_BlockSearch : Bool;   // Block search active / Recherche de blocs active
      E_M30 : Bool;   // M2/M30 active / M2/M30 actif
      E_Transform : Bool;   // Transformation active
      E_ProgTest : Bool;   // Program test active / Test de programme actif
      E_OEMChan : Byte;   // OEM channel signals feedback / Signalisation en retour signaux de canal OEM
      E_ProgRunning : Bool;   // Program running / Programme en cours d'exécution
      E_ProgWait : Bool;   // Program waiting / Programme en attente
      E_ProgStop : Bool;   // Program stopped / Programme arrêté
      E_ProgInterrupt : Bool;   // Program interrupted / Programme interrompu
      E_ProgAborted : Bool;   // Program aborted / Programme abandonné
      E_ChanActive : Bool;   // Channel active / Canal actif
      E_ChanInterrupt : Bool;   // Channel interrupted / Canal interrompu
      E_ChanReset : Bool;   // Channel reset / Reset canal
      E_StartReq : Bool;   // Start request / Demande de démarrage
      E_StopReq : Bool;   // Stop request / Demande d'arrêt
      E_AxesRef : Bool;   // All axes referenced / Référencer tous les axes
      E_AxesStop : Bool;   // All axes stationary / Tous les axes à l'arrêt
      E_IR_Activ : Bool;   // Interrupt processing active / Traitement d'interruption actif
      E_ChanRO : Bool;   // Channel ready for operation / Canal prêt à fonctionner
      E_NCKalarmChan : Bool;   // Channel-specific NCK alarm present / Alarme NCK spécifique à un canal présente
      E_NCKalarmStop : Bool;   // NCK alarm with processing stop present / Alarme NCK avec d'arrêt d'usinage présente
      E_CHW1 : Bool;   // Contour handwheel 1 on / Manivelle de contour 1
      E_CHW2 : Bool;   // Contour handwheel 2 on / Manivelle de contour 2
      E_CHW3 : Bool;   // Contour handwheel 3 on / Manivelle de contour 3
      E_CLC : Bool;   // CLC active / CLC actif
      E_CLCStopLL : Bool;   // CLC stopped lower limit / CLC arrêté limite inférieure
      E_CLCStopUL : Bool;   // CLC stopped upper limit / CLC arrêté limite supérieure
      E_RIEnabIgnored : Bool;   // Read-in enable is ignored / Activation Charger ignorée
      E_StopBlkEndSBLsuppr : Bool;   // Stop at block end with SBL is suppressed / Inhiber arrêt sur fin de bloc avec SBL
      E_StrokeEA : Bool;   // Stroke release active / Déblocage course actif
      E_AcknManStrokEnab : Bool;   // Acknowledgment of manual stroke release / Acquittement déblocage manuel de course
      f38_2 : Bool;
      f38_3 : Bool;
      f38_4 : Bool;
      f38_5 : Bool;
      f38_6 : Bool;
      f38_7 : Bool;
      E_ProtZoneNOK : Bool;   // Protection zones not guaranteed / Zones de protection non garanties
      E_NCalarmWithProgStop : Bool;   // NC alarm with program stop / Alarme CN avec arrêt du programme
      f39_2 : Bool;
      E_ReducedDynamicsActive : Bool;   // Reduced dynamics mode is active / Le mode de dynamique réduite est actif
      E_SblStopAtBlockEnd : Bool;   // Stop at block end due to single block / Arrêt en fin de bloc en raison du mode bloc par bloc
      E_InvCHWDirOfRot : Bool;   // Contour handwheel direction of rotation invert actively / Inversion active du sens de rotation manivelle de contour
      E_CfgStopFuncActive : Bool;   // Configured stop function is activated / La fonction d'arrêt configuré est activée
      E_CfgStopAtBlockEnd : Bool;   // Stop at block end due to configured stop / Arrêt en fin de bloc en raison de l'arrêt configuré
      E_Geo : Array[1..3] of Struct   // Status signals of geometry axis [1..3] / Signaux d'état de l'axe géométrique [1..3]
         HW1 : Bool;   // Handwheel 1 active / Manivelle 1 active
         HW2 : Bool;   // Handwheel 2 active / Manivelle 2 active
         HW3 : Bool;   // Handwheel 3 active / Manivelle 3 active
         f0_3 : Bool;
         TReqMinus : Bool;   // Travel requests minus / Demandes de déplacement moins
         TReqPlus : Bool;   // Travel requests plus / Demandes de déplacement plus
         TCMinus : Bool;   // Traverse command minus / Instruction de déplacement moins
         TCPlus : Bool;   // Traverse command plus / Instruction de déplacement plus
         INC1 : Bool;   // INC 1 active
         INC10 : Bool;   // INC 10 active
         INC100 : Bool;   // INC 100 active
         INC1000 : Bool;   // INC 1000 active
         INC10000 : Bool;   // INC 10000 active
         INCVar : Bool;   // INC variable active / Variable INC active
         ContManTravelAct : Bool;   // Continuous manual travel active / Mode manuel continu actif
         f1_7 : Bool;
         OEM : Byte;   // OEM signals / Signaux OEM
         InvHWDirOfRot : Bool;   // Handwheel direction of rotation invert actively / Inverser activement sens manivelle
         f3_1 : Bool;
         f3_2 : Bool;
         f3_3 : Bool;
         f3_4 : Bool;
         f3_5 : Bool;
         f3_6 : Bool;
         f3_7 : Bool;
         f4 : Byte;
      END_STRUCT;
      M1Change : Bool;   // M function 1 change / Fonction M 1 modification
      M2Change : Bool;   // M function 2 change / Fonction M 2 modification
      M3Change : Bool;   // M function 3 change / Fonction M 3 modification
      M4Change : Bool;   // M function 4 change / Fonction M 4 modification
      M5Change : Bool;   // M function 5 change / Fonction M 5 modification
      f58_5 : Bool;
      f58_6 : Bool;
      f58_7 : Bool;
      M1NDec : Bool;   // M function 1 not decoded / Fonction M 1 non décodée
      M2NDec : Bool;   // M function 2 not decoded / Fonction M 2 non décodée
      M3NDec : Bool;   // M function 3 not decoded / Fonction M 3 non décodée
      M4NDec : Bool;   // M function 4 not decoded / Fonction M 4 non décodée
      M5NDec : Bool;   // M function 5 not decoded / Fonction M 5 non décodée
      f59_5 : Bool;
      f59_6 : Bool;
      f59_7 : Bool;
      S1Change : Bool;   // S function 1 change / Fonction S 1 modification
      S2Change : Bool;   // S function 2 change / Fonction S 2 modification
      S3Change : Bool;   // S function 3 change / Fonction S 3 modification
      f60_3 : Bool;
      S1Quick : Bool;   // S function 1 quick / Fonction S 1 rapide
      S2Quick : Bool;   // S function 2 quick / Fonction S 2 rapide
      S3Quick : Bool;   // S function 3 quick / Fonction S 3 rapide
      f60_7 : Bool;
      T1Change : Bool;   // T function 1 change / Fonction T 1 modification
      T2Change : Bool;   // T function 2 change / Fonction T 2 modification
      T3Change : Bool;   // T function 3 change / Fonction T 3 modification
      f61_3 : Bool;
      T1Quick : Bool;   // T function 1 quick / Fonction T 1 rapide
      T2Quick : Bool;   // T function 2 quick / Fonction T 2 rapide
      T3Quick : Bool;   // T function 3 quick / Fonction T 3 rapide
      f61_7 : Bool;
      D1Change : Bool;   // D function 1 change / Fonction D 1 modification
      D2Change : Bool;   // D function 2 change / Fonction D 2 modification
      D3Change : Bool;   // D function 3 change / Fonction D 3 modification
      f62_3 : Bool;
      D1Quick : Bool;   // D function 1 quick / Fonction D 1 rapide
      D2Quick : Bool;   // D function 2 quick / Fonction D 2 rapide
      D3Quick : Bool;   // D function 3 quick / Fonction D 3 rapide
      f62_7 : Bool;
      EChange : Bool;   // E function change / Fonction E modification
      f63_1 : Bool;
      f63_2 : Bool;
      f63_3 : Bool;
      EQuick : Bool;   // E function quick / Fonction E rapide
      f63_5 : Bool;
      f63_6 : Bool;
      f63_7 : Bool;
      H1Change : Bool;   // H function 1 change / Fonction H 1 modification
      H2Change : Bool;   // H function 2 change / Fonction H 2 modification
      H3Change : Bool;   // H function 3 change / Fonction H 3 modification
      f64_3 : Bool;
      H1Quick : Bool;   // H function 1 quick / Fonction H 1 rapide
      H2Quick : Bool;   // H function 2 quick / Fonction H 2 rapide
      H3Quick : Bool;   // H function 3 quick / Fonction H 3 rapide
      f64_7 : Bool;
      F1Change : Bool;   // F function 1 change / Fonction F 1 modification
      F2Change : Bool;   // F function 2 change / Fonction F 2 modification
      F3Change : Bool;   // F function 3 change / Fonction F 3 modification
      F4Change : Bool;   // F function 4 change / Fonction F 4 modification
      F5Change : Bool;   // F function 5 change / Fonction F 5 modification
      F6Change : Bool;   // F function 6 change / Fonction F 6 modification
      f65_6 : Bool;
      f65_7 : Bool;
      M1Quick : Bool;   // M function 1 quick / Fonction M 1 rapide
      M2Quick : Bool;   // M function 2 quick / Fonction M 2 rapide
      M3Quick : Bool;   // M function 3 quick / Fonction M 3 rapide
      M4Quick : Bool;   // M function 4 quick / Fonction M 4 rapide
      M5Quick : Bool;   // M function 5 quick / Fonction M 5 rapide
      f66_5 : Bool;
      f66_6 : Bool;
      f66_7 : Bool;
      F1Quick : Bool;   // F function 1 quick / Fonction F 1 rapide
      F2Quick : Bool;   // F function 2 quick / Fonction F 2 rapide
      F3Quick : Bool;   // F function 3 quick / Fonction F 3 rapide
      F4Quick : Bool;   // F function 4 quick / Fonction F 4 rapide
      F5Quick : Bool;   // F function 5 quick / Fonction F 5 rapide
      F6Quick : Bool;   // F function 6 quick / Fonction F 6 rapide
      f67_6 : Bool;
      f67_7 : Bool;
      ExtM1 : Int;   // Extended address M function 1 (16 bit INT) / Fonction M à adresse étendue 1 (16 bits INT)
      M1 : DInt;   // M function 1 (DInt) / Fonction M 1 (DInt)
      ExtM2 : Int;   // Extended address M function 1 (16 bit INT) / Fonction M à adresse étendue 1 (16 bits INT)
      M2 : DInt;   // M function 2 (DInt) / Fonction M 2 (DInt)
      ExtM3 : Int;   // Extended address M function 1 (16 bit INT) / Fonction M à adresse étendue 1 (16 bits INT)
      M3 : DInt;   // M function 3 (DInt) / Fonction M 3 (DInt)
      ExtM4 : Int;   // Extended address M function 1 (16 bit INT) / Fonction M à adresse étendue 1 (16 bits INT)
      M4 : DInt;   // M function 4 (DInt) / Fonction M 4 (DInt)
      ExtM5 : Int;   // Extended address M function 1 (16 bit INT) / Fonction M à adresse étendue 1 (16 bits INT)
      M5 : DInt;   // M function 5 (DInt) / Fonction M 5 (DInt)
      ExtS1 : Int;   // Extended address S function 1 (16 bit INT) / Fonction S à adresse étendue 1 (16 bits INT)
      S1 : Real;   // S function 1 (REAL) / Fonction S 1 (REAL)
      ExtS2 : Int;   // Extended address S function 2 (16 bit INT) / Fonction S à adresse étendue 2 (16 bits INT)
      S2 : Real;   // S function 2 (REAL) / Fonction S 2 (REAL)
      ExtS3 : Int;   // Extended address S function 3 (16 bit INT) / Fonction S à adresse étendue 3 (16 bits INT)
      S3 : Real;   // S function 3 (REAL) / Fonction S 3 (REAL)
      ExtT1 : Int;   // Extended address T function 1 (16 bit INT)T : DINT; //T function (DInt)f122 : INT;f124 : INT;f126 : INT; //Change in case of 8-digit T function / Fonction T à adresse étendue 1 (16 Bit INT)T : DINT; //fonction T (DInt)f122 : INT;f124 : INT;f126 : INT; //Modifier pour une fonction T à 8 chiffres
      T1 : Int;   // T function 1 (INT) / Fonction T 1 (INT)
      ExtT2 : Int;   // Extended address T function 2 (16 bit INT) / Fonction T à adresse étendue 2 (16 bits INT)
      T2 : Int;   // T function 2 (INT) / Fonction T 2 (INT)
      ExtT3 : Int;   // Extended address T function 3 (16 bit INT) / Fonction T à adresse étendue 3 (16 bits INT)
      T3 : Int;   // T function 3 (INT) / Fonction T 3 (INT)
      ExtD1 : Byte;   // Extended address D function 1 (8 bit INT)D : INT;f132 : INT; //Change in case of 5-digit D function / Fonction D à adresse étendue 1 (8 bits INT)D : INT;f132 : INT; //Modifier pour une fonction D à 5 chiffres
      D1 : Byte;   // D function 1 (8 bit INT) / Fonction D 1 (8 bits INT)
      ExtD2 : Byte;   // Extended address D function 2 (8 bit INT) / Fonction D à adresse étendue 2 (8 bits INT)
      D2 : Byte;   // D function 2 (8 bit INT) / Fonction D 2 (8 bits INT)
      ExtD3 : Byte;   // Extended address D function 3 (8 bit INT) / Fonction D à adresse étendue 3 (8 bits INT)
      D3 : Byte;   // D function 3 (8 bit INT) / Fonction D 3 (8 bits INT)
      ExtE : Int;   // Extended address D function 3 (16 bit INT) / Fonction D à adresse étendue 3 (16 bits INT)
      "E" : Real;   // E function (REAL) / Fonction E (REAL)
      ExtH1 : Int;   // Extended address H function 1 (16 bit INT) / Fonction H à adresse étendue 1 (16 bits INT)
      H1 : Real;   // H function 1 (REAL), DInt also in DBD396 / Fonction H 1 (REAL), DInt également dans DBD396
      ExtH2 : Int;   // Extended address H function 2 (16 bit INT) / Fonction H à adresse étendue 2 (16 bits INT)
      H2 : Real;   // H function 2 (REAL), DInt also in DBD400 / Fonction H 2 (REAL), DInt également dans DBD400
      ExtH3 : Int;   // Extended address H function 3 (16 bit INT) / Fonction H à adresse étendue 3 (16 bits INT)
      H3 : Real;   // H function 3 (REAL), DInt also in DBD404 / Fonction H 3 (REAL), DInt également dans DBD404
      ExtF1 : Int;   // Extended address F function 1 (16 bit INT) / Fonction F à adresse étendue 1 (16 bits INT)
      F1 : Real;   // F function 1 (REAL) / Fonction F 1 (REAL)
      ExtF2 : Int;   // Extended address F function 2 (16 bit INT) / Fonction F à adresse étendue 2 (16 bits INT)
      F2 : Real;   // F function 2 (REAL) / Fonction F 2 (REAL)
      ExtF3 : Int;   // Extended address F function 3 (16 bit INT) / Fonction F à adresse étendue 3 (16 bits INT)
      F3 : Real;   // F function 3 (REAL) / Fonction F 3 (REAL)
      ExtF4 : Int;   // Extended address F function 4 (16 bit INT) / Fonction F à adresse étendue 4 (16 bits INT)
      F4 : Real;   // F function 4 (REAL) / Fonction F 4 (REAL)
      ExtF5 : Int;   // Extended address F function 5 (16 bit INT) / Fonction F à adresse étendue 5 (16 bits INT)
      F5 : Real;   // F function 5 (REAL) / Fonction F 5 (REAL)
      ExtF6 : Int;   // Extended address F function 6 (16 bit INT) / Fonction F à adresse étendue 6 (16 bits INT)
      F6 : Real;   // F function 6 (REAL) / Fonction F 6 (REAL)
      MDyn : Array[0..99] of Bool;   // Dynamic M functions [0..99] / Fonctions M dynamiques [0..99]
      GAct : Array[1..64] of Byte;   // Active G function of group [1..64] / Fonction G active du groupe [1..64]
      E_MRPactivated : Array[1..10] of Bool;   // Machine-related protection zone [1..10] preactivated / Zone de protection référencée dans le SCM [1..10] préactivé
      E_CSPactivated : Array[1..10] of Bool;   // Channel-specific protection zone [1..10] preactivated / Zone de protection spécifique au canal [1..10] préactivée
      E_MRPViolated : Array[1..10] of Bool;   // Machine-related protection zone [1..10] violated / Zone de protection référencée dans le SCM [1..10] dépassée
      E_CSPViolated : Array[1..10] of Bool;   // Channel-specific protection zone [1..10] violated from P4 on / Zone de protection spécifique au canal [1..10] dépassée à partir de P4
      f_280_0 : Bool;
      A_Str_Synon : Bool;   // Request of syn.action to NCK / Demande d'action synchrone vers NCK
      f_280_2 : Bool;
      f_280_3 : Bool;
      f_280_4 : Bool;
      f_280_5 : Bool;
      f_280_6 : Bool;
      f_280_7 : Bool;
      f_281_0 : Bool;
      A_Str_Synfrom : Bool;   // Request syn.action from NCK / Demande d'action synchrone depuis NCK
      f_281_2 : Bool;
      f_281_3 : Bool;
      f_281_4 : Bool;
      f_281_5 : Bool;
      f_281_6 : Bool;
      f_281_7 : Bool;
      f_282 : Int;
      f_284 : Int;
      f_286 : Int;
      f_288 : Int;
      f_290 : Int;
      f_292 : Int;
      f_294 : Int;
      f_296 : Int;
      f_298 : Int;
      A_SynDisabl : Array[1..64] of Bool;   // Disable synchronous actions / Désactiver actions synchrones
      E_SynDisabled : Array[1..64] of Bool;   // Synchronous actions disabled / Actions synchrones désactivées
      E_G00 : Bool;   // Active G functions / Fonctions G actives
      f316_1 : Bool;
      f316_2 : Bool;
      f316_3 : Bool;
      f316_4 : Bool;
      f316_5 : Bool;
      f316_6 : Bool;
      f316_7 : Bool;
      E_ExtLang : Bool;   // External language mode active / Mode de langage externe actif
      E_WS_Setp : Bool;   // Workpiece setpoint reached / Consigne pièce atteinte
      f317_2 : Bool;
      f317_3 : Bool;
      f317_4 : Bool;
      E_DriveTest : Bool;   // Travel request drive test / Demande de déplacement test d'entraînement
      E_PTP_Travel : Bool;   // PTP travel active / Déplacement PTP actif
      E_ToolMissing : Bool;   // Tool missing / Outil manquant
      E_ASUP_Stop : Bool;   // ASUP stopped / ASUP arrêté
      E_SearchAct : Bool;   // Search active / Recherche active
      E_TOFF : Bool;   // TOFF active / TOFF actif
      E_TOFFmovem : Bool;   // TOFF motion active / Déplacement TOFF actif
      E_StopDelayed : Bool;   // Stop delayed / Arrêt temporisé
      E_AssM01 : Bool;   // Associated M01 active / M01 associé actif
      E_DRY : Bool;   // Dry-run feedrate active / Marche d'essai avance active
      E_Overstore : Bool;   // Overstore active / Overstore actif
      E_REPOS_EdgeAckn : Bool;   // REPOS MODE EDGE ACKN
      E_REPOS_PMode0 : Bool;   // REPOS Path Mode Ackn 0
      E_REPOS_PMode1 : Bool;   // REPOS Path Mode Ackn 1
      E_REPOS_PMode2 : Bool;   // REPOS Path Mode Ackn 2
      E_DelayFTS : Bool;   // Delay FTS / Temporisation FTS
      E_REPOS_DEFERRA : Bool;   // REPOS DEFERRA L Chan
      E_Stop_NoDelayR : Bool;   // Stop-delay area not accepted / Plage de temporisation d'arrêt non acceptée
      E_NoToolChangeCmd : Bool;   // No tool change command active / Aucun ordre de changement d'outil actif
      A_Ori : Array[1..3] of Struct   // Control signals for orientation axes [1..3] / Signaux de commande pour axes d'orientation [1..3]
         HW1 : Bool;   // Activate handwheel 1 / Activer manivelle 1
         HW2 : Bool;   // Activate handwheel 2 / Activer manivelle 2
         HW3 : Bool;   // Activate handwheel 3 / Activer manivelle 3
         FDStop : Bool;   // Feedrate stop / Arrêt avance
         Disabl : Bool;   // Traversing key lock / Verrouiller touche de déplacement
         RapidTrOR : Bool;   // Rapid traverse override / Correction marche rapide
         Minus : Bool;   // Traversing key minus / Touche de déplacement moins
         Plus : Bool;   // Traversing key plus / Touche de déplacement plus
         INC1 : Bool;   // INC 1 active
         INC10 : Bool;   // INC 10 active
         INC100 : Bool;   // INC 100 active
         INC1000 : Bool;   // INC 1000 active
         INC10000 : Bool;   // INC 10000 active
         INCVar : Bool;   // INC variable active / Variable INC active
         OEM : Byte;   // OEM signals / Signaux OEM
         InvHWDirOfRot : Bool;   // Inverting handwheel direction of rotation / Inverser sens de rotation manivelle
         f3_1 : Bool;
         f3_2 : Bool;
         f3_3 : Bool;
         f3_4 : Bool;
         f3_5 : Bool;
         f3_6 : Bool;
         f3_7 : Bool;
      END_STRUCT;
      E_Ori : Array[1..3] of Struct   // Control signals for orientation axes [1..3] / Signaux de commande pour axes d'orientation [1..3]
         HW1 : Bool;   // Handwheel 1 active / Manivelle 1 active
         HW2 : Bool;   // Handwheel 2 active / Manivelle 2 active
         HW3 : Bool;   // Handwheel 3 active / Manivelle 3 active
         f0_3 : Bool;
         TReqMinus : Bool;   // Travel requests minus / Demandes de déplacement moins
         TReqPlus : Bool;   // Travel requests plus / Demandes de déplacement plus
         TCMinus : Bool;   // Traverse command minus / Instruction de déplacement moins
         TCPlus : Bool;   // Traverse command plus / Instruction de déplacement plus
         INC1 : Bool;   // INC 1 active
         INC10 : Bool;   // INC 10 active
         INC100 : Bool;   // INC 100 active
         INC1000 : Bool;   // INC 1000 active
         INC10000 : Bool;   // INC 10000 active
         INCVar : Bool;   // INC variable active / Variable INC active
         OEM : Byte;   // OEM signals / Signaux OEM
         InvHWDirOfRot : Bool;   // Handwheel direction of rotation invert actively / Inverser activement sens manivelle
         f3_1 : Bool;
         f3_2 : Bool;
         f3_3 : Bool;
         f3_4 : Bool;
         f3_5 : Bool;
         f3_6 : Bool;
         f3_7 : Bool;
      END_STRUCT;
      E_TPrewarnLimit : Bool;   // Tool prewarn limit reached / Seuil de préavis outil atteint
      E_TLimit : Bool;   // Tool limit reached / Limite d'outil atteinte
      E_TNewRepl : Bool;   // Transition to new replacement tool / Transition vers nouvel outil de remplacement
      E_TLastRepl : Bool;   // Last replacement tool of the tool group / Dernier outil de remplacement du groupe d'outils
      f344_4 : Bool;
      f344_5 : Bool;
      f344_6 : Bool;
      f344_7 : Bool;
      f345 : Byte;
      f346 : Byte;
      f347 : Byte;
      E_TNoPrewarnLimit : DInt;   // T number for tool prewarn limit / Numéro d'outil pour seuil de préavis outil
      E_TNoLimit : DInt;   // T number for tool limit / Numéro d'outil pour limite d'outil
      E_TNoNewRepl : DInt;   // T number of the new replacement tool / Numéro d'outil du nouvel outil de remplacement
      E_TNoLastRepl : DInt;   // T number of the last replacement tool / Numéro d'outil du dernier outil de remplacement
      E_Cycle_Sig : Array[0..15] of Bool;   // Cycles input signals / Signaux d'entrée des cycles
      A_Cycle_Sig : Array[0..15] of Bool;   // Cycles output signals / Signaux de sortie des cycles
      E_OEM_TechnoSig : Array[0..31] of Bool;   // OEM Techno input signals / Signaux d'entrée techno OEM
      A_OEM_TechnoSig : Array[0..31] of Bool;   // OEM Techno output signals / Signaux de sortie techno OEM
      E_ProgEvent_Start : Bool;   // Active Prog-Event: Start / Prog-Event actif : Démarrage
      E_ProgEvent_M30 : Bool;   // Active Prog-Event: M30 / Prog-Event actif : M30
      E_ProgEvent_Reset : Bool;   // Active Prog-Event: Start / Prog-Event actif : Démarrage
      E_ProgEvent_PowerOn : Bool;   // Active Prog-Event: Power on / Prog-Event actif : Mise sous tension
      E_ProgEvent_SearchRun : Bool;   // Active Prog-Event: Search / Prog-Event actif : Recherche
      f376_5 : Bool;
      f376_6 : Bool;
      f376_7 : Bool;
      E_CollCheckStop : Bool;   // Stop of Collision Check / Arrêt du contrôle de collision
      E_StopCondition : Bool;   // Stop Condition / Condition d'arrêt
      f377_2 : Bool;
      f377_3 : Bool;
      E_JogRetract : Bool;   // JOG Retract active / Retrait JOG actif
      E_RetractData : Bool;   // Retract data available / Données de retrait disponibles
      E_JOG_Circles : Bool;   // JOG in circles / JOG en cercles
      f377_7 : Bool;
      E_AnyAsup : Bool;   // AnyASUP activ / AnyASUP actif
      E_SilentAsup : Bool;   // Silent ASUP active / ASUP silencieux actif
      f378_2 : Bool;
      f378_3 : Bool;
      f378_4 : Bool;
      f378_5 : Bool;
      f378_6 : Bool;
      f378_7 : Bool;
      f379 : Byte;
      f380 : Array[0..31] of Bool;   // Reserved / Réservé
      A_ProgJump : Bool;   // Control program jump / Saut programme de commande
      f384_1 : Bool;
      f384_2 : Bool;
      f384_3 : Bool;
      f384_4 : Bool;
      f384_5 : Bool;
      f384_6 : Bool;
      f384_7 : Bool;
      A_InKeyG1 : Bool;   // Grinding signal 1 / Signal rectification 1
      A_InKeyG2 : Bool;   // Grinding signal 2 / Signal rectification 2
      A_InKeyG3 : Bool;   // Grinding signal 3 / Signal rectification 3
      A_InKeyG4 : Bool;   // Grinding signal 4 / Signal rectification 4
      A_InKeyG5 : Bool;   // Grinding signal 5 / Signal rectification 5
      A_InKeyG6 : Bool;   // Grinding signal 6 / Signal rectification 6
      A_InKeyG7 : Bool;   // Grinding signal 7 / Signal rectification 7
      A_InKeyG8 : Bool;   // Grinding signal 8 / Signal rectification 8
      A_InKeyGEn1 : Bool;   // Enable grinding signal 1 / Activer signal rectification 1
      A_InKeyGEn2 : Bool;   // Enable grinding signal 2 / Activer signal rectification 2
      A_InKeyGEn3 : Bool;   // Enable grinding signal 3 / Activer signal rectification 3
      A_InKeyGEn4 : Bool;   // Enable grinding signal 4 / Activer signal rectification 4
      A_InKeyGEn5 : Bool;   // Enable grinding signal 5 / Activer signal rectification 5
      A_InKeyGEn6 : Bool;   // Enable grinding signal 6 / Activer signal rectification 6
      A_InKeyGEn7 : Bool;   // Enable grinding signal 7 / Activer signal rectification 7
      A_InKeyGEn8 : Bool;   // Enable grinding signal 8 / Activer signal rectification 8
      A_InKeyGRunIn1 : Bool;   // Run grinding function 1 / Exécuter fonction de rectification 1
      A_InKeyGRunIn2 : Bool;   // Run grinding function 2 / Exécuter fonction de rectification 2
      A_InKeyGRunIn3 : Bool;   // Run grinding function 3 / Exécuter fonction de rectification 3
      A_InKeyGRunIn4 : Bool;   // Run grinding function 4 / Exécuter fonction de rectification 4
      A_InKeyGRunIn5 : Bool;   // Run grinding function 5 / Exécuter fonction de rectification 5
      A_InKeyGRunIn6 : Bool;   // Run grinding function 6 / Exécuter fonction de rectification 6
      A_InKeyGRunIn7 : Bool;   // Run grinding function 7 / Exécuter fonction de rectification 7
      A_InKeyGRunIn8 : Bool;   // Run grinding function 8 / Exécuter fonction de rectification 8
      E_TransformNo : Byte;   // Active transformation number / Numéro de la transformation active
      f389 : Byte;
      E_InKeyGIsEn1 : Bool;   // Grinding signal 1 enabled / Signal rectification 1 activé
      E_InKeyGIsEn2 : Bool;   // Grinding signal 2 enabled / Signal rectification 2 activé
      E_InKeyGIsEn3 : Bool;   // Grinding signal 3 enabled / Signal rectification 3 activé
      E_InKeyGIsEn4 : Bool;   // Grinding signal 4 enabled / Signal rectification 4 activé
      E_InKeyGIsEn5 : Bool;   // Grinding signal 5 enabled / Signal rectification 5 activé
      E_InKeyGIsEn6 : Bool;   // Grinding signal 6 enabled / Signal rectification 6 activé
      E_InKeyGIsEn7 : Bool;   // Grinding signal 7 enabled / Signal rectification 7 activé
      E_InKeyGIsEn8 : Bool;   // Grinding signal 8 enabled / Signal rectification 8 activé
      E_InKeyGRunOut1 : Bool;   // NCK status of grinding function 1 / État NCK fonction de rectification 1
      E_InKeyGRunOut2 : Bool;   // NCK status of grinding function 3 / État NCK fonction de rectification 3
      E_InKeyGRunOut3 : Bool;   // NCK status of grinding function 3 / État NCK fonction de rectification 3
      E_InKeyGRunOut4 : Bool;   // NCK status of grinding function 4 / État NCK fonction de rectification 4
      E_InKeyGRunOut5 : Bool;   // NCK status of grinding function 5 / État NCK fonction de rectification 5
      E_InKeyGRunOut6 : Bool;   // NCK status of grinding function 6 / État NCK fonction de rectification 6
      E_InKeyGRunOut7 : Bool;   // NCK status of grinding function 7 / État NCK fonction de rectification 7
      E_InKeyGRunOut8 : Bool;   // NCK status of grinding function 8 / État NCK fonction de rectification 8
      E_CART_JOG_MODE : Byte;   // Coordinate system for Cartesian jog traverse / Système de coordonnées pour déplacement cartésien en mode JOG
      f393 : Byte;
      f394 : Byte;
      f395 : Byte;
      H1_DInt : DInt;   // H Function 1 (DInt) / Fonction H 1 (DInt)
      H2_DInt : DInt;   // H Function 2 (DInt) / Fonction H 2 (DInt)
      H3_DInt : DInt;   // H Function 3 (DInt) / Fonction H 3 (DInt)
      E_AxisSelType : Byte;   // 0: MachAxis, 1: GeoAxis
      E_AxisSelAxis : Byte;   // Axis number / Numéro d'axe
      E_AxisSelRequest : Bool;   // Axis selection (touch) / Sélection d'axe (touche)
      f410_1 : Bool;
      f410_2 : Bool;
      f410_3 : Bool;
      f410_4 : Bool;
      f410_5 : Bool;
      f410_6 : Bool;
      f410_7 : Bool;
      f411 : Byte;
      A_AxisSelTypeActive : Byte;   // 0: MachAxis, 1: GeoAxis (return) / 0: MachAxis, 1: GeoAxis (retour)
      A_AxisSelAxisActive : Byte;   // Axis number (return) / Numéro d'axe (retour)
   END_STRUCT;
   // // A_Geo[2].HW1 : Activate handwheel 1 / Activer manivelle 1
   // // A_Geo[3].HW1 : Activate handwheel 1 / Activer manivelle 1
   // // A_Geo[2].HW2 : Activate handwheel 2 / Activer manivelle 2
   // // A_Geo[3].HW2 : Activate handwheel 2 / Activer manivelle 2
   // // A_Geo[2].HW3 : Activate handwheel 3 / Activer manivelle 3
   // // A_Geo[3].HW3 : Activate handwheel 3 / Activer manivelle 3
   // // A_Geo[2].FDStop : Feedrate stop / Arrêt avance
   // // A_Geo[3].FDStop : Feedrate stop / Arrêt avance
   // // A_Geo[2].Disabl : Traversing key disable / Désactiver la touche de déplacement
   // // A_Geo[3].Disabl : Traversing key disable / Désactiver la touche de déplacement
   // // A_Geo[2].RapidTrOR : Rapid traverse override / Correction marche rapide
   // // A_Geo[3].RapidTrOR : Rapid traverse override / Correction marche rapide
   // // A_Geo[2].Minus : Traversing key minus / Touche de déplacement moins
   // // A_Geo[3].Minus : Traversing key minus / Touche de déplacement moins
   // // A_Geo[2].Plus : Traversing key plus / Touche de déplacement plus
   // // A_Geo[3].Plus : Traversing key plus / Touche de déplacement plus
   // // A_Geo[2].INC1 : INC 1
   // // A_Geo[3].INC1 : INC 1
   // // A_Geo[2].INC10 : INC 10
   // // A_Geo[3].INC10 : INC 10
   // // A_Geo[2].INC100 : INC 100
   // // A_Geo[3].INC100 : INC 100
   // // A_Geo[2].INC1000 : INC 1000
   // // A_Geo[3].INC1000 : INC 1000
   // // A_Geo[2].INC10000 : INC 10000
   // // A_Geo[3].INC10000 : INC 10000
   // // A_Geo[2].INCVar : INC variable / Variable INC
   // // A_Geo[3].INCVar : INC variable / Variable INC
   // // A_Geo[2].ContManTravel : Continuous manual travel / Mode manuel continu
   // // A_Geo[3].ContManTravel : Continuous manual travel / Mode manuel continu
   // // A_Geo[2].OEM : OEM signals / Signaux OEM
   // // A_Geo[3].OEM : OEM signals / Signaux OEM
   // // A_Geo[2].InvHWDirOfRot : Invert handwheel direction of rotation / Inverser sens de rotation manivelle
   // // A_Geo[3].InvHWDirOfRot : Invert handwheel direction of rotation / Inverser sens de rotation manivelle
   // // A_Geo[1] : Control signals for geometry axis [1..3] / Signaux de commande pour axe géométrique [1..3]
   // // A_Geo[2] : Control signals for geometry axis [1..3] / Signaux de commande pour axe géométrique [1..3]
   // // A_Geo[3] : Control signals for geometry axis [1..3] / Signaux de commande pour axe géométrique [1..3]
   // // E_Geo[2].HW1 : Handwheel 1 active / Manivelle 1 active
   // // E_Geo[3].HW1 : Handwheel 1 active / Manivelle 1 active
   // // E_Geo[2].HW2 : Handwheel 2 active / Manivelle 2 active
   // // E_Geo[3].HW2 : Handwheel 2 active / Manivelle 2 active
   // // E_Geo[2].HW3 : Handwheel 3 active / Manivelle 3 active
   // // E_Geo[3].HW3 : Handwheel 3 active / Manivelle 3 active
   // // E_Geo[2].TReqMinus : Travel requests minus / Demandes de déplacement moins
   // // E_Geo[3].TReqMinus : Travel requests minus / Demandes de déplacement moins
   // // E_Geo[2].TReqPlus : Travel requests plus / Demandes de déplacement plus
   // // E_Geo[3].TReqPlus : Travel requests plus / Demandes de déplacement plus
   // // E_Geo[2].TCMinus : Traverse command minus / Instruction de déplacement moins
   // // E_Geo[3].TCMinus : Traverse command minus / Instruction de déplacement moins
   // // E_Geo[2].TCPlus : Traverse command plus / Instruction de déplacement plus
   // // E_Geo[3].TCPlus : Traverse command plus / Instruction de déplacement plus
   // // E_Geo[2].INC1 : INC 1 active
   // // E_Geo[3].INC1 : INC 1 active
   // // E_Geo[2].INC10 : INC 10 active
   // // E_Geo[3].INC10 : INC 10 active
   // // E_Geo[2].INC100 : INC 100 active
   // // E_Geo[3].INC100 : INC 100 active
   // // E_Geo[2].INC1000 : INC 1000 active
   // // E_Geo[3].INC1000 : INC 1000 active
   // // E_Geo[2].INC10000 : INC 10000 active
   // // E_Geo[3].INC10000 : INC 10000 active
   // // E_Geo[2].INCVar : INC variable active / Variable INC active
   // // E_Geo[3].INCVar : INC variable active / Variable INC active
   // E_Geo[1].ContManTravelAct := false;
   // // E_Geo[2].ContManTravelAct : Continuous manual travel active / Mode manuel continu actif
   // // E_Geo[3].ContManTravelAct : Continuous manual travel active / Mode manuel continu actif
   // E_Geo[1].f1_7 := false;
   // // E_Geo[2].OEM : OEM signals / Signaux OEM
   // // E_Geo[3].OEM : OEM signals / Signaux OEM
   // // E_Geo[2].InvHWDirOfRot : Handwheel direction of rotation invert actively / Inverser activement sens manivelle
   // // E_Geo[3].InvHWDirOfRot : Handwheel direction of rotation invert actively / Inverser activement sens manivelle
   // // E_Geo[1] : Status signals of geometry axis [1..3] / Signaux d'état de l'axe géométrique [1..3]
   // // E_Geo[2] : Status signals of geometry axis [1..3] / Signaux d'état de l'axe géométrique [1..3]
   // // E_Geo[3] : Status signals of geometry axis [1..3] / Signaux d'état de l'axe géométrique [1..3]
   // // A_Ori[2].HW1 : Activate handwheel 1 / Activer manivelle 1
   // // A_Ori[3].HW1 : Activate handwheel 1 / Activer manivelle 1
   // // A_Ori[2].HW2 : Activate handwheel 2 / Activer manivelle 2
   // // A_Ori[3].HW2 : Activate handwheel 2 / Activer manivelle 2
   // // A_Ori[2].HW3 : Activate handwheel 3 / Activer manivelle 3
   // // A_Ori[3].HW3 : Activate handwheel 3 / Activer manivelle 3
   // // A_Ori[2].FDStop : Feedrate stop / Arrêt avance
   // // A_Ori[3].FDStop : Feedrate stop / Arrêt avance
   // // A_Ori[2].Disabl : Traversing key lock / Verrouiller touche de déplacement
   // // A_Ori[3].Disabl : Traversing key lock / Verrouiller touche de déplacement
   // // A_Ori[2].RapidTrOR : Rapid traverse override / Correction marche rapide
   // // A_Ori[3].RapidTrOR : Rapid traverse override / Correction marche rapide
   // // A_Ori[2].Minus : Traversing key minus / Touche de déplacement moins
   // // A_Ori[3].Minus : Traversing key minus / Touche de déplacement moins
   // // A_Ori[2].Plus : Traversing key plus / Touche de déplacement plus
   // // A_Ori[3].Plus : Traversing key plus / Touche de déplacement plus
   // // A_Ori[2].INC1 : INC 1 active
   // // A_Ori[3].INC1 : INC 1 active
   // // A_Ori[2].INC10 : INC 10 active
   // // A_Ori[3].INC10 : INC 10 active
   // // A_Ori[2].INC100 : INC 100 active
   // // A_Ori[3].INC100 : INC 100 active
   // // A_Ori[2].INC1000 : INC 1000 active
   // // A_Ori[3].INC1000 : INC 1000 active
   // // A_Ori[2].INC10000 : INC 10000 active
   // // A_Ori[3].INC10000 : INC 10000 active
   // // A_Ori[2].INCVar : INC variable active / Variable INC active
   // // A_Ori[3].INCVar : INC variable active / Variable INC active
   // // A_Ori[2].OEM : OEM signals / Signaux OEM
   // // A_Ori[3].OEM : OEM signals / Signaux OEM
   // // A_Ori[2].InvHWDirOfRot : Inverting handwheel direction of rotation / Inverser sens de rotation manivelle
   // // A_Ori[3].InvHWDirOfRot : Inverting handwheel direction of rotation / Inverser sens de rotation manivelle
   // // A_Ori[1] : Control signals for orientation axes [1..3] / Signaux de commande pour axes d'orientation [1..3]
   // // A_Ori[2] : Control signals for orientation axes [1..3] / Signaux de commande pour axes d'orientation [1..3]
   // // A_Ori[3] : Control signals for orientation axes [1..3] / Signaux de commande pour axes d'orientation [1..3]
   // // E_Ori[2].HW1 : Handwheel 1 active / Manivelle 1 active
   // // E_Ori[3].HW1 : Handwheel 1 active / Manivelle 1 active
   // // E_Ori[2].HW2 : Handwheel 2 active / Manivelle 2 active
   // // E_Ori[3].HW2 : Handwheel 2 active / Manivelle 2 active
   // // E_Ori[2].HW3 : Handwheel 3 active / Manivelle 3 active
   // // E_Ori[3].HW3 : Handwheel 3 active / Manivelle 3 active
   // // E_Ori[2].TReqMinus : Travel requests minus / Demandes de déplacement moins
   // // E_Ori[3].TReqMinus : Travel requests minus / Demandes de déplacement moins
   // // E_Ori[2].TReqPlus : Travel requests plus / Demandes de déplacement plus
   // // E_Ori[3].TReqPlus : Travel requests plus / Demandes de déplacement plus
   // // E_Ori[2].TCMinus : Traverse command minus / Instruction de déplacement moins
   // // E_Ori[3].TCMinus : Traverse command minus / Instruction de déplacement moins
   // // E_Ori[2].TCPlus : Traverse command plus / Instruction de déplacement plus
   // // E_Ori[3].TCPlus : Traverse command plus / Instruction de déplacement plus
   // // E_Ori[2].INC1 : INC 1 active
   // // E_Ori[3].INC1 : INC 1 active
   // // E_Ori[2].INC10 : INC 10 active
   // // E_Ori[3].INC10 : INC 10 active
   // // E_Ori[2].INC100 : INC 100 active
   // // E_Ori[3].INC100 : INC 100 active
   // // E_Ori[2].INC1000 : INC 1000 active
   // // E_Ori[3].INC1000 : INC 1000 active
   // // E_Ori[2].INC10000 : INC 10000 active
   // // E_Ori[3].INC10000 : INC 10000 active
   // // E_Ori[2].INCVar : INC variable active / Variable INC active
   // // E_Ori[3].INCVar : INC variable active / Variable INC active
   // // E_Ori[2].OEM : OEM signals / Signaux OEM
   // // E_Ori[3].OEM : OEM signals / Signaux OEM
   // // E_Ori[2].InvHWDirOfRot : Handwheel direction of rotation invert actively / Inverser activement sens manivelle
   // // E_Ori[3].InvHWDirOfRot : Handwheel direction of rotation invert actively / Inverser activement sens manivelle
   // // E_Ori[1] : Control signals for orientation axes [1..3] / Signaux de commande pour axes d'orientation [1..3]
   // // E_Ori[2] : Control signals for orientation axes [1..3] / Signaux de commande pour axes d'orientation [1..3]
   // // E_Ori[3] : Control signals for orientation axes [1..3] / Signaux de commande pour axes d'orientation [1..3]
END_TYPE

TYPE "LBP_typeConfigData"
TITLE = Configuration parameter / Paramètre de configuration
// User data type for block LBP_ConfigData [DB7] / Type de données utilisateur pour bloc LBP_ConfigData [DB7]
   STRUCT
      MCPNum : Int;   // Inputs starting here / Début des entrées
      MCP1In : Struct   // Pointer / Pointeur
         DBNo : Word;
         Addr : DWord;
      END_STRUCT;
      MCP1Out : Struct   // Pointer / Pointeur
         DBNo : Word;
         Addr : DWord;
      END_STRUCT;
      reservedByte14_25 : Array[14..25] of Byte;
      MCP1BusAdr : Int := 6;
      MCP1Timeout : S5Time := S5T#700MS;
      reservedByte30_31 : Array[30..31] of Byte;
      MCP2In : Struct   // Pointer / Pointeur
         DBNo : Word;
         Addr : DWord;
      END_STRUCT;
      MCP2Out : Struct   // Pointer / Pointeur
         DBNo : Word;
         Addr : DWord;
      END_STRUCT;
      reservedByte44_55 : Array[44..55] of Byte;
      MCP2BusAdr : Int;
      MCP2Timeout : S5Time := S5T#700MS;
      reservedByte60_61 : Array[60..61] of Byte;
      reservedBool62_0 : Bool;
      MCP1Stop : Bool;
      MCP2Stop : Bool;
      MCP1NotSend : Bool;
      MCP2NotSend : Bool;
      reservedBool62_5 : Bool;
      reservedBool62_6 : Bool;
      MCPBusType : Byte := BYTE#16#05;
      HTIf : Int;
      HTIn : Struct   // Pointer / Pointeur
         DBNo : Word;
         Addr : DWord;
      END_STRUCT;
      HTOut : Struct   // Pointer / Pointeur
         DBNo : Word;
         Addr : DWord;
      END_STRUCT;
      reservedByte78_95 : Array[78..95] of Byte;
      HTAdr : Int := 2;
      reservedByte98_107 : Array[98..107] of Byte;
      reservedBool108_0 : Bool;
      HTStop : Bool;
      HTNotSend : Bool;
      NCCyclTimeout : S5Time := S5T#200MS;
      NCRunupTimeout : S5Time := S5T#50S;
      ListMDecGrp : Int;
      reservedBool116_0 : Bool;
      MMCToIF : Bool := TRUE;
      HWheelMMC : Bool := TRUE;
      reservedBool116_3 : Bool;
      MCP_IF_TCS : Bool;
      ExtendChanAxMsg : Bool;
      HMIAxisSel : Bool;
      DeactivateCtrlEnergy : Bool;
      MsgUser : Int := 10;
      reservedBool120_0 : Bool;
      IRAuxfuT : Bool;
      IRAuxfuH : Bool;
      IRAuxfuE : Bool;
      UserVersion : Struct   // Pointer / Pointeur
         DBNo : Word;
         Addr : DWord;
      END_STRUCT;
      OpKeyNum : Int;
      Op1KeyIn : Struct   // Pointer / Pointeur
         DBNo : Word;
         Addr : DWord;
      END_STRUCT;
      Op1KeyOut : Struct   // Pointer / Pointeur
         DBNo : Word;
         Addr : DWord;
      END_STRUCT;
      Op1KeyBusAdr : Int;
      Op2KeyIn : Struct   // Pointer / Pointeur
         DBNo : Word;
         Addr : DWord;
      END_STRUCT;
      Op2KeyOut : Struct   // Pointer / Pointeur
         DBNo : Word;
         Addr : DWord;
      END_STRUCT;
      Op2KeyBusAdr : Int;
      Op1KeyStop : Bool;
      Op2KeyStop : Bool;
      Op1KeyNotSend : Bool;
      Op2KeyNotSend : Bool;
      reservedByte159 : Byte;
      IdentMcpBusAdr : Int;
      IdentMcpProfilNo : Byte;
      IdentMcpBusType : Byte := BYTE#16#05;
      IdentMcpStrobe : Bool;
      MaxModeGroup : Int;   // Outputs starting here / Début des sorties
      MaxChan : Int;
      MaxAxis : Int;
      ActiveChan : Array[1..10] of Bool;
      ActiveAxis : Array[1..31] of Bool;
      MaxNumUserDataInt : Int;
      MaxNumUserDataHex : Int;
      MaxNumUserDataReal : Int;
      IdentMcpType : Byte;
      IdentMcpLengthIn : Byte;
      IdentMcpLengthOut : Byte;
      reservedByte188_199 : Array[188..199] of Byte;   // Static starting here / Début statique
      LBPVersionInfo : String[44];
      UserVersionInfo : String[44];
      GenerateAlarmMsgs : Struct
         NumActAlarmMsgs : UInt;
         Error : Bool;
         StatusID : UInt;
         Status : Word;
      END_STRUCT;
      OpUnitCommId : UInt := 1;   // ID for OpUnitComm / ID pour OpUnitComm
      OpUnitInterfaceId : HW_ANY := 262;   // Hardware identifier of Ethernet interface for OpUnitComm / Identifiant matériel de l'interface Ethernet pour OpUnitComm
      MCP1ConnectionId : CONN_OUC := 1001;   // Connection identifier for MCP 1 / Identifiant de connexion pour MCP 1
      MCP2ConnectionId : CONN_OUC := 1002;   // Connection identifier for MCP 2 / Identifiant de connexion pour MCP 2
      HTConnectionId : CONN_OUC := 1003;   // Connection identifier for handheld unit / Identifiant de connexion pour terminal portatif
      Op1KeyConnectionId : CONN_OUC := 1004;   // Connection identifier for Direct Key 1 / Identifiant de connexion pour Direct Key 1
      Op2KeyConnectionId : CONN_OUC := 1005;   // Connection identifier for Direct Key 2 / Identifiant de connexion pour Direct Key 2
      IdentConnectionId : CONN_OUC := 1006;   // Connection identifier for identification / Identifiant de connexion pour identification
      MCP1LocalUdpPort : UInt := 16001;   // Local UDP port for MCP 1 / Port UDP local pour MCP 1
      MCP2LocalUdpPort : UInt := 16002;   // Local UDP port for MCP 2 / Port UDP local pour MCP 2
      HTLocalUdpPort : UInt := 16003;   // Local UDP port for handheld unit / Port UDP local pour unité de commande portable
      Op1KeyLocalUdpPort : UInt := 16004;   // Local UDP port for Direct Key 1 / Port UDP local pour Direct Key 1
      Op2KeyLocalUdpPort : UInt := 16005;   // Local UDP port for Direct Key 2 / Port UDP local pour Direct Key 2
      IdentLocalUdpPort : UInt := 16006;   // Local UDP port for Ident / Port UDP local pour Ident
      MCP1Error : Bool;   // Error MCP 1 / Erreur MCP 1
      MCP1Status : Word;   // Error information MCP 1 / Information erreur MCP 1
      MCP2Error : Bool;   // Error MCP 2 / Erreur MCP 2
      MCP2Status : Word;   // Error information MCP 2 / Information erreur MCP 2
      HTError : Bool;   // Error handheld unit / Erreur terminal portatif
      HTStatus : Word;   // Error information handheld unit / Information erreur terminal portatif
      Op1KeyError : Bool;   // Error Direct Key 1 / Erreur Direct Key 1
      Op1KeyStatus : Word;   // Error information Direct Key 1 / Information erreur Direct Key 1
      Op2KeyError : Bool;   // Error Direct Key 2 / Erreur Direct Key 2
      Op2KeyStatus : Word;   // Error information Direct Key 2 / Information erreur Direct Key 2
      IdentError : Bool;   // Error identification / Identification d'erreur
      IdentStatus : Word;   // Error information Identification / Identification d'erreur Identification
      MCP1Ready : Bool;   // MCP1 connected / MCP1 connecté
      MCP2Ready : Bool;   // MCP2 connected / MCP2 connecté
      HTReady : Bool;   // Handheld unit connected / Terminal portatif connecté
      Op1KeyReady : Bool;   // Direct Key 1 connected / Direct Key 1 connecté
      Op2KeyReady : Bool;   // Direct Key 2 connected / Direct Key 2 connecté
   END_STRUCT;
END_TYPE

